(* CODESYS project Mk5 Aorta.library
   DefaultNamespace: _AORTA_
   Company: Atlas Copco
   Version: 2.0.0.0
   Title: Mk5 Aorta
   Author: Peter

Project tree, tasks and I/O mapping:
  libraries: Mk5 Definitions, 2.0.0.0 (Atlas Copco); Standard, * (System); SysMem, * (System); Mk5 Blackfin Libraries, 2.0.0.0 (Atlas Copco); Mk5 CANOpen Driver Interfaces, 2.0.0.0 (Atlas Copco); Mk5 CANOpen Driver Full, 2.0.0.0 (Atlas Copco); Mk5 IO and Protection System Interfaces, 2.0.0.0 (Atlas Copco); Mk5 Special IVL, 2.0.0.0 (Atlas Copco); Mk5 Lookup Tables Interfaces, 2.0.0.0 (Atlas Copco); Mk5 Display Texts Touch, 2.0.0.0 (Atlas Copco); Mk5 Drives Interfaces, 2.0.0.0 (Atlas Copco); Mk5 Tools Base Full, 2.0.0.0 (Atlas Copco); Mk5 CondensationPoint Interfaces, 2.0.0.0 (Atlas Copco); Mk5 Dryers Handler Interfaces, 2.0.0.0 (Atlas Copco); Mk5 Dryers Base Interfaces, 2.0.0.0 (Atlas Copco); Mk5 Retain Interfaces, 2.0.0.0 (Atlas Copco); Mk5 Special Functions interfaces, 2.0.0.0 (Atlas Copco); Mk5 StatusInfo Interfaces, 2.0.0.0 (Atlas Copco); Mk5 System Root, 2.0.0.0 (Atlas Copco); Mk5 Aorta Interfaces, 2.0.0.0 (Atlas Copco); Mk5 OD Interfaces, 2.0.0.0 (Atlas Copco); Mk5s Display Helpers Interfaces, 2.0.0.0 (Atlas Copco); Mk5s Display Base, 2.0.0.0 (Atlas Copco); Mk5s Display Definitions, 2.0.0.0 (Atlas Copco); Mk5 IO and Protection System Full, 2.0.0.0 (Atlas Copco); Mk5 CondensationPoint Full, 2.0.0.0 (Atlas Copco); Util, 3.5.18.0 (System); Mk5 SpeedControl Interfaces, 2.0.0.0 (Atlas Copco); Mk5 Display Constants, 2.0.0.0 (Atlas Copco); Mk5 ProtecSpec_Comon, 2.0.0.0 (Atlas Copco)
  Aorta/
    PrimaStuff/
      function block fbtCANOpenDriver_Aorta_Prima [ST]: mxInit, prpxValidData
      function block fbtAorta_Prima [ST]: mxInit, mxEnable, mxReset, mxResetCANOpenDriver, mxRun, mxPosition, mxHoming, mxDumpHomingSettings, prpxEnabled, mxWriteValue, prpdwPosition, mxConfigurationError
    Driver/
      CANOpenDriver/
        function block fbtCANOpenDriver_Aorta_Tri [ST]: mxInit, prpxValidData
        PDO Topic/
          Rx/
            function block fbtAorta_SW [ST]: prpx_2_OperationEnabled, prpx_0_ReadyToSwitchOn, prpx_5_QuickStop, prpx_9_Remote, prpx_4_VoltageEnabled, prpx_6_SwitchOnDisabled, prpx_12_SetpointInProcess, prpx_1_SwitchedOn, prpx_7_Warning, prpx_10_TargetReached, prpx_3_Fault, mbState
            function block fbtAorta_ActualPosition [ST]: prpdwPosition
            function block fbtAorta_ActualOperationMode [ST]: prpxHoming
            function block fbtAorta_ActualPosition_2Bytes [ST]: prpdwPosition
            function block fbtAorta_Alarm [ST]: prpwAlarm
            function block fbtAorta_SW_Trinamics [ST]: prpx_02_OperationEnabled, prpx_00_ReadyToSwitchOn, prpx_05_QuickStop, prpx_09_Remote, prpx_04_VoltageEnabled, prpx_06_SwitchOnDisabled, prpx_12_SetpointInProcess, prpx_01_SwitchedOn, prpx_07_Warning, prpx_10_TargetReached, prpx_03_Fault, mbState, prpx_14_MotorActive, prpx_15_Direction_Down, prpx_12_HomingMode_HomeAttained
            function block fbtAorta_ActualPosition_1 [ST]: prpdwPosition
          Tx/
            function block fbtAorta_CW [ST]: prpx_1_EnableVoltage, prpx_3_EnableOperation, prpx_0_SwitchOn, prpx_4_NewSetpoint, prpx_7_FaultReset, prpx_2_NoQuickStop, prpx_6_Relative, mxDisableOperation, mxShutDown
            function block fbtAorta_OperationMode [ST]: prpxHoming
            function block fbtAorta_HomingMode [ST]: prpbMode
            function block fbtAorta_TargetPosition [ST]: prpdwPosition
            function block fbtAorta_TargetPosition_2Bytes [ST]: prpdwPosition
            function block fbtAorta_Dummy_2Bytes [ST]: prpdwPosition
      function block fbtAorta_Trinamics [ST]: mxInit, mxPosition, dwMicroStepsMoved, mxHoming, mxReadStrokeLength, mxReadVendorID, prpxEnabled, mxEnable, mxReset, mxDisable, mxSettings, prpdwPosition, mxDumpSettings, mxCollectData, prpitfCANOpenDriver, mxForcedNMTReset, prpdiPCBTemp, prpdiHousingTemp, mxConfigurationError, prpwSW, prpdwError11Count, prpdwRequiredPosition, prpxDirection
      Settings/
        function block fbtAorta_AllSettings_Tri [ST]: mxInit, mxGetSDO
        function block fbtAorta_AllSettings_Pri [ST]: mxAdd, mxGetSDO, mxInit
      data type DS302_States
      data type Aorta_StateMachine
      data type Aorta_Errors
      data type Aorta_CycleStates
    AortaEngine/
      data type STR_Error
      function block fbtAortaSettingsDownloader [ST]: mxDownload, prpbActiveSubIndex, prpbStatus, prpxBusy, mxInit, prppDownloadError
      data type ENUM_AortaEngine_StateMain
      data type ENUM_AortaEngine_StateHoming
      data type ENUM_AortaEngine_StateOperating
      data type ENUM_AortaEngine_StateRetract
      function block fbtAortaEngine_Base [ST]: mxInit_SysPyLog, mxInit, mxInit_Output, mxLoadSettings, mxRun, mxHoming, mxOperating, mxEnable, mxRetract, mdiNextPosition, prppdiDebugPosition, prppdiDebugStroke_FullSteps, prppdiDebugStroke_MicroSteps, prppdiDebugStroke_Rotations, prppdiDebugError, prppdiDebugErrorPosition, prppdiDebugMicroStepsInMove, prppdiDebugRotDirection, prppdiDebugStallDetectPosition, prppdiDebugStallRetractDelta, prppdiDebugStallRetractPosition, prppdiStatusWord, prppdiDebugError11Counter, prpdwPosition, prpwError, mReset, mxOD3000Define, mxConfigurationError, prprLimitedPosition, prpxActive, prpxFixedPositionActive, prpxHomingActive, mxStartHoming, mxMoveToFixedPosition, prpdwHomingStrokeMS, prpxCANDriverError, mxCollectInfoSDO3000
      global variables GVL_AORTA
      data type ENUM_TimeUnit
      data type ENUM_AortaDownloader_States
      IVL/
        function block fbtIVL_STCPosition [ST]: mxIVL_Settings_Overwrite
    Special Alarm/
      function block fbtProtecSpec_STCValve [ST]: mxInitSpecial, mxLoadSettings, mwCheckProtection, prpitfProtectionInfo, prpxMoreInfo, mxReset, mxResolveMPLLinks
      function block fbtProtecSpec_STCValve_Info [ST]: mxGetMk5sData, mxSetMk5sData, mInit
  CoolPower/
    CANOpenDriver/
      function block fbtCANOpenDriver_CoolPower [ST]: mxInit, mxConfigPrep, mxSetAddress_NT, mxResetAddress
      function block fbtSDO_Series_CoolPower [ST]: mxGetSDO, mxInitList, prpbAddress
    PDO Topic/
      Rx/
        function block fbtCoolPower_ActualOperationMode [ST]: prpbOperationMode
        function block fbtCoolPower_ActualVelocity [ST]: prpdwVelocity
        function block fbtCoolPower_ActualPosition [ST]: prpdwPosition
        function block fbtCoolPower_SW [ST]: prpx_2_OperationEnabled, prpx_0_ReadyToSwitchOn, prpx_5_QuickStop, prpx_9_Remote, prpx_4_VoltageEnabled, prpx_6_SwitchOnDisabled, prpx_12_OMS1, prpx_1_SwitchedOn, prpx_7_Warning, prpx_10_TargetReached, prpx_3_Fault, mbState, prpx_8_Synchronized, prpx_11_InternalLimitActive, prpx_13_OMS2, prpx_15_ClosedLoop
        function block fbtCoolPower_DigitalInputs [ST]: mxGetInput
        function block fbtCoolPower_MaxMotorSpeed [ST]: prpdwMaxSpeed
        function block fbtCoolPower_RunningHours [ST]: prpdwRunningHours
        function block fbtCoolPower_SerialNumber_1_6 [ST]: prpdwSerial_1_6
        function block fbtCoolPower_SerialNumber_7_11 [ST]: prpdwSerial_7_11
      Tx/
        function block fbtCoolPower_CW [ST]: prpx_1_EnableVoltage, prpx_3_EnableOperation, prpx_0_SwitchOn, prpx_4_OMS1, prpx_7_FaultReset, prpx_2_NoQuickStop, prpx_8_Halt, prpx_5_OMS2, prpx_6_OMS3, prpx_9_OMS4
        function block fbtCoolPower_OperationMode [ST]: prpbOperationMode
        function block fbtCoolPower_TargetVelocity [ST]: prpdwVelocity
        function block fbtCoolPower_TargetPosition [ST]: prpdwPosition
        function block fbtCoolPower_DriveSubMode [ST]: prpx_0_ClosedLoop, prpx_1_VoS, prpx_2_Brake, prpx_3_CurrentReduction, prpx_5_Torque, prpx_6_BLDC
        function block fbtCoolPower_ProfileVelocity [ST]: prpdwVelocity
        function block fbtCoolPower_DigitalOutputs [ST]: mxSetOutput
      global variables GVL_NanoTecAddresses
    function block fbtCoolPower_NanoTec [ST]: prpbOperationMode, prpdwMaxSpeed, prpdwRunningHours, prpdwSpeed, prpulSerialNumber, prpxHalt, prpxIsOperational, prpbModel, prpdwTotalHours, mxDisable, mxEnable, mxInit, mxRun, mxReadOut, mxConfigure, mxReset, mxClean, mxResetCounter
  Oil Free Air/
    Offset/
      function block fbtOffsetsConditionalSetpointCalculation [ST]: mxInit, mxCollectInfoSDO3000, mxOD3000Define, mxRun, mxGetValueOffset
      function block fbtOffset [ST]: prprValue, mxGetInput, mxInit, prpbInputNumber, mxGetSubIndex, prpxZeroValue, mxGetPowerValue
    Conditional Setpoint/
      function block fbtConditionalSetpointCalculation [ST]: mxInit, mxInit_Output, mxRun, mxOD3000Define, mxCollectInfoSDO3000
      function block fbtInput_CondSetpoint_ERSetpoint [ST]: mxInit_ER, mxGetInput, prpxSwitchToER
      function block fbtIVL_CondSetpointTemp [ST]: mxSetOutput, prpwSDO, mxInit, prpbOffsetNumber, prpbOffsetNumberER, mxIVL_Settings_Overwrite
    Energy Recovery Regulation/
      function block fbtEnergyRecoveryRegulation [ST]: prprEnergyRecoverySetpointTemperature, mxInit, mxRun, prpxSwitchToER, mxOD3000Define, mxInit_Output
      data type ENUM_HeatQualityOffset
      function block fbtIVL_ERSetpointTemp [ST]: mxIVL_Settings_Overwrite
  Handler/
    function block fbtSTCHandler [ST]: mxGetSTCValve, mxInit, mxInit_Output, mxOD3000Define, mxRun, mxGetOptimalSERCalculation
  Industrial Air SER Calculation/
    function block fbtOptimalSERCalculation [ST]: mxInit, mxLoadSettings, mRun, prpiTemperature, prppdiDebugTemperature, mxInit_Output
    function block fbtIVL_OptimalSERTemp [ST]: mxIVL_Settings_Overwrite
*)

// Aorta/Driver/DS302_States
{attribute 'qualified_only'}
{attribute 'strict'}
TYPE DS302_States :
(
	bNoInfo,
	bNotReadyToSwitchOn,
	bSwitchOnDisabled,
	bReadyToSwitchOn,
	bSwitchedOn,
	bOperationEnabled,
	bQuickStopActive,
	bFault,
	bFaultReactionActive,
	bUnknown_Error,
	bWaitforReset
)BYTE;
END_TYPE

// Aorta/Driver/Aorta_StateMachine
{attribute 'qualified_only'}
{attribute 'strict'}
TYPE Aorta_StateMachine :
(
	bStart,
	bFlank,
	bFinish,
	bWait,
	bReadStroke,
	bMotorActive
)BYTE;
END_TYPE

// Aorta/Driver/Aorta_Errors
{attribute 'qualified_only'}
{attribute 'strict'}
TYPE Aorta_Errors :
(
	NoError							:= 0,
	Initiate_StartupTimeout			:= 1,
	Initiate_Fault					:= 2,
	Initiate_DumpSettings			:= 3,
	
	Homing_NotEnabled				:= 4,
	Homing_TimeOut					:= 5,
	Homing_FailedToGetStrokeLength	:= 6,
	Homing_RangeTooSmall			:= 7,
// 	Homing_Failed					:= 8,

	Position_NotEnabled				:= 9,
	Position_Stall					:= 10,
	Position_TimeOut				:= 11,
	Position_Retract				:= 12,
	Position_PI_Error				:= 13,
	STCValve_Active_No_Alarm		:= 14,
	CAN_Out							:= 100,
	StuckInErrorState				:= 101
)	BYTE
	:= NoError;
END_TYPE

// Aorta/Driver/Aorta_CycleStates
{attribute 'qualified_only'}
{attribute 'strict'}
TYPE Aorta_CycleStates :
(
	Idle,
	Send,
	TimeOut,
	StallDetected,
	StallHandling
	
);
END_TYPE

// Aorta/AortaEngine/STR_Error
TYPE STR_Error :
STRUCT
	tDelay			: TIME;
	tonDelay		: TON;
	bNotification	: BYTE;
END_STRUCT
END_TYPE

// Aorta/AortaEngine/ENUM_AortaEngine_StateMain
{attribute 'qualified_only'}
{attribute 'strict'}
TYPE ENUM_AortaEngine_StateMain :
(
	Enable,
	Homing,
	Operating,
	Retract,
	Reset,
	Error,
	CAN_Error,
	Valve_detached
);
END_TYPE

// Aorta/AortaEngine/ENUM_AortaEngine_StateHoming
{attribute 'qualified_only'}
{attribute 'strict'}
TYPE ENUM_AortaEngine_StateHoming :
(
	Start,
	Home,
	CheckRange,
	Retry
);
END_TYPE

// Aorta/AortaEngine/ENUM_AortaEngine_StateOperating
{attribute 'qualified_only'}
{attribute 'strict'}
TYPE ENUM_AortaEngine_StateOperating :
(
	GoToPosition,
	SetNextPosition,
	Wait
);
END_TYPE

// Aorta/AortaEngine/ENUM_AortaEngine_StateRetract
{attribute 'qualified_only'}
{attribute 'strict'}
TYPE ENUM_AortaEngine_StateRetract :
(
	SetRetractPosition,
	Retract
);
END_TYPE

// Aorta/AortaEngine/ENUM_TimeUnit
{attribute 'qualified_only'}
// {attribute 'strict'}
TYPE ENUM_TimeUnit :
(
	Millisecond	:= 0,
	Second		:= 1,
	Minute		:= 2,
	Hour		:= 3,
	Day			:= 4
)	BYTE;
END_TYPE

// Aorta/AortaEngine/ENUM_AortaDownloader_States
{attribute 'qualified_only'}
TYPE ENUM_AortaDownloader_States :
(
	findtype,
	select,
	download
);
END_TYPE

// Oil Free Air/Energy Recovery Regulation/ENUM_HeatQualityOffset
{attribute 'qualified_only'}
{attribute 'strict'}
TYPE ENUM_HeatQualityOffset :
(
	Not_used := 0,
	Input_IO,
	Minimal, 
	Medium, 
	Maximal	
	
)BYTE;
END_TYPE

// CoolPower/PDO Topic/GVL_NanoTecAddresses
{attribute 'qualified_only'}
VAR_GLOBAL CONSTANT
	SerialNumber1_6_Index 		: WORD := 16#2410;
	SerialNumber1_6_Subindex 	: BYTE := 1;
	SerialNumber7_11_Index 		: WORD := 16#2410;
	SerialNumber7_11_Subindex 	: BYTE := 2;
	RunningHours_Index			: WORD := 16#2410;
	RunningHours_Subindex		: BYTE := 3;
	TotalHours_Index			: WORD := 16#2410;
	TotalHours_Subindex			: BYTE := 4;
	MaxSpeed_Index				: WORD := 16#6080;
	MaxSpeed_Subindex			: BYTE := 0;
	Model_Index					: WORD := 16#2410;
	Model_Subindex				: BYTE := 5;
END_VAR

// Aorta/AortaEngine/GVL_AORTA
{attribute 'qualified_only'}
VAR_GLOBAL
	wControlRange 			: WORD := 10000;
	wControlRange01Percent 	: WORD := 1;  // same as above, but 0.1%
END_VAR

// Aorta/Driver/CANOpenDriver/PDO Topic/Tx/fbtAorta_CW
FUNCTION_BLOCK fbtAorta_CW EXTENDS fbtPDO_Word 
VAR_INPUT
END_VAR
VAR_OUTPUT
END_VAR
VAR
END_VAR

PROPERTY prpx_1_EnableVoltage : BOOL
SET
wData.1:=prpx_1_EnableVoltage;
END_SET
END_PROPERTY

PROPERTY prpx_3_EnableOperation : BOOL
SET
wData.3:=prpx_3_EnableOperation;
END_SET
END_PROPERTY

PROPERTY prpx_0_SwitchOn : BOOL
SET
wData.0:=prpx_0_SwitchOn;
END_SET
END_PROPERTY

PROPERTY prpx_4_NewSetpoint : BOOL
SET
wData.4:=prpx_4_NewSetpoint;
END_SET
END_PROPERTY

PROPERTY prpx_7_FaultReset : BOOL
SET
wData.7:=prpx_7_FaultReset;
END_SET
END_PROPERTY

PROPERTY prpx_2_NoQuickStop : BOOL
SET
wData.2:=prpx_2_NoQuickStop;
END_SET
END_PROPERTY

PROPERTY prpx_6_Relative : BOOL
SET
wData.6:=prpx_6_Relative;
END_SET
END_PROPERTY

METHOD mxDisableOperation : BOOL
VAR_INPUT
END_VAR
wData:=7;
END_METHOD

METHOD mxShutDown : BOOL
VAR_INPUT
END_VAR
wData:=6; //Shutdown aorta valve
END_METHOD

END_FUNCTION_BLOCK

// Aorta/Driver/CANOpenDriver/PDO Topic/Rx/fbtAorta_SW
FUNCTION_BLOCK fbtAorta_SW EXTENDS fbtPDO_Word 
VAR_INPUT
END_VAR
VAR_OUTPUT
END_VAR
VAR
END_VAR

PROPERTY prpx_2_OperationEnabled : BOOL
GET
prpx_2_OperationEnabled:=wData.2;
END_GET
END_PROPERTY

PROPERTY prpx_0_ReadyToSwitchOn : BOOL
GET
prpx_0_ReadyToSwitchOn:=wData.0;
END_GET
END_PROPERTY

PROPERTY prpx_5_QuickStop : BOOL
GET
prpx_5_QuickStop:=wData.5;
END_GET
END_PROPERTY

PROPERTY prpx_9_Remote : BOOL
GET
prpx_9_Remote:=wData.9;
END_GET
END_PROPERTY

PROPERTY prpx_4_VoltageEnabled : BOOL
GET
prpx_4_VoltageEnabled:=wData.4;
END_GET
END_PROPERTY

PROPERTY prpx_6_SwitchOnDisabled : BOOL
GET
prpx_6_SwitchOnDisabled:=wData.6;
END_GET
END_PROPERTY

PROPERTY prpx_12_SetpointInProcess : BOOL
GET
prpx_12_SetpointInProcess:=wData.12;
END_GET
END_PROPERTY

PROPERTY prpx_1_SwitchedOn : BOOL
GET
prpx_1_SwitchedOn:=wData.1;
END_GET
END_PROPERTY

PROPERTY prpx_7_Warning : BOOL
GET
prpx_7_Warning:=wData.7;
END_GET
END_PROPERTY

PROPERTY prpx_10_TargetReached : BOOL
GET
prpx_10_TargetReached:=wData.10;
END_GET
END_PROPERTY

PROPERTY prpx_3_Fault : BOOL
GET
prpx_3_Fault:=wData.3;
END_GET
END_PROPERTY

METHOD mbState : BYTE
VAR_INPUT
END_VAR
VAR
	wTmp : WORD;
END_VAR
wTmp := wData AND 16#000F;
CASE wTmp OF
0 : IF wData.6 THEN // wSW.prpx_6_SwitchOnDisabled 
		mbState := DS302_States.bSwitchOnDisabled;
	ELSE
		mbState := DS302_States.bNotReadyToSwitchOn;
	END_IF

1 : IF wData.5=1 AND wData.6=0 THEN
		mbState:= DS302_States.bReadyToSwitchOn;	
	ELSE
		mbState:=DS302_States.bUnknown_Error;
	END_IF

3 : IF wData.5=1 AND wData.6=0 THEN
		mbState:= DS302_States.bSwitchedOn;	
	ELSE
		mbState:=DS302_States.bUnknown_Error;
	END_IF

7 : IF wData.5=1 AND wData.6=0 THEN
		mbState:= DS302_States.bOperationEnabled;	
	ELSIF wData.5=0 AND wData.6=0 THEN
		mbState:= DS302_States.bQuickStopActive;	
	ELSE
		mbState:=DS302_States.bUnknown_Error;
	END_IF

8 : IF wData.6=0 THEN
		mbState:= DS302_States.bFault;	
	ELSE
		mbState:=DS302_States.bUnknown_Error;
	END_IF
		
16#F : IF wData.6=0 THEN
		mbState:= DS302_States.bFaultReactionActive;	
	ELSE
		mbState:=DS302_States.bUnknown_Error;
	END_IF
ELSE // case
			mbState:=DS302_States.bUnknown_Error;
END_CASE
END_METHOD

END_FUNCTION_BLOCK

// Aorta/Driver/CANOpenDriver/fbtCANOpenDriver_Aorta_Tri
FUNCTION_BLOCK fbtCANOpenDriver_Aorta_Tri EXTENDS fbtCANOpenDriver_Base
VAR_INPUT
END_VAR
VAR_OUTPUT
END_VAR
VAR
END_VAR

METHOD mxInit : BOOL
VAR_INPUT
	bCANAddress  			: BYTE;
END_VAR
eDriverState:=CAN_StateMachine.Idle;
bTheAddress := bCANAddress;

fbNMTCommands.mxInit(bAddress := bCANAddress);
END_METHOD

PROPERTY prpxValidData : BOOL
GET
prpxValidData:=TRUE;
END_GET
END_PROPERTY

END_FUNCTION_BLOCK

// Aorta/Driver/CANOpenDriver/PDO Topic/Tx/fbtAorta_OperationMode
FUNCTION_BLOCK fbtAorta_OperationMode EXTENDS fbtPDO_Byte
VAR_INPUT
END_VAR
VAR_OUTPUT
END_VAR
VAR
//	bMode : BYTE := 1;
END_VAR

PROPERTY prpxHoming : BOOL
SET
IF prpxHoming THEN
	bData := 6;
ELSE
	bData := 1; // pp
END_IF
END_SET
END_PROPERTY

END_FUNCTION_BLOCK

// Aorta/Driver/CANOpenDriver/PDO Topic/Tx/fbtAorta_HomingMode
FUNCTION_BLOCK fbtAorta_HomingMode EXTENDS fbtPDO_Byte
VAR_INPUT
END_VAR
VAR_OUTPUT
END_VAR
VAR
END_VAR

PROPERTY prpbMode : BYTE
SET
bData := prpbMode;
END_SET
END_PROPERTY

END_FUNCTION_BLOCK

// Aorta/Driver/CANOpenDriver/PDO Topic/Tx/fbtAorta_TargetPosition
FUNCTION_BLOCK fbtAorta_TargetPosition EXTENDS fbtPDO_DWORD
VAR_INPUT
END_VAR
VAR_OUTPUT
END_VAR
VAR
//	dwPosition : DWORD;
END_VAR

PROPERTY prpdwPosition : DWORD
SET
dwData := prpdwPosition;
END_SET
GET
prpdwPosition := dwData;
END_GET
END_PROPERTY

END_FUNCTION_BLOCK

// Aorta/Driver/CANOpenDriver/PDO Topic/Rx/fbtAorta_ActualPosition
FUNCTION_BLOCK fbtAorta_ActualPosition EXTENDS fbtPDO_DWORD
VAR_INPUT
END_VAR
VAR_OUTPUT
END_VAR
VAR
//	dwPosition : DWORD;
END_VAR

PROPERTY prpdwPosition : DWORD
GET
prpdwPosition:=dwData;
END_GET
END_PROPERTY

END_FUNCTION_BLOCK

// Aorta/Driver/CANOpenDriver/PDO Topic/Rx/fbtAorta_ActualOperationMode
FUNCTION_BLOCK fbtAorta_ActualOperationMode EXTENDS fbtPDO_Byte
VAR_INPUT
END_VAR
VAR_OUTPUT
END_VAR
VAR
//	bMode : BYTE := 1;
END_VAR

PROPERTY prpxHoming : BOOL
GET
IF bData = 6 THEN
	prpxHoming:=TRUE;
ELSE
	prpxHoming:=FALSE;
END_IF
END_GET
END_PROPERTY

END_FUNCTION_BLOCK

// Aorta/Driver/fbtAorta_Trinamics
FUNCTION_BLOCK fbtAorta_Trinamics
VAR
	bMyCANAddress			: BYTE;
	xStartLocal				: BOOL;
	
	fbCANOpen 				: fbtCANOpenDriver_Aorta_Tri;

	// dwBrand					: DWORD;
	
	Aorta_CW 				: fbtAorta_CW;
	Aorta_OperationMode 	: fbtAorta_OperationMode;
	Aorta_HomingMode 		: fbtAorta_HomingMode;
	Aorta_TargetPosition 	: fbtAorta_TargetPosition; 

	Aorta_SW				: fbtAorta_SW_Trinamics;
	Aorta_ActualPosition	: fbtAorta_ActualPosition;
	Aorta_ActualMode		: fbtAorta_ActualOperationMode;

	PCBTemp 				: fbtPDO_DWORD;
	HousingTemp             : fbtPDO_DWORD;

	wDownloadState			: WORD;
	xDownloadStart			: BOOL;
	wDownloadStateWait		: TON;
	
	Tp_CommandTimeOut		: TP;
	xStartTimeOut			: BOOL;
	bDriveState				: BYTE;
	
	bstate	 				: BYTE;
// position cycle
//	CycleTime 				: TON;
//	CycleState				: Aorta_CycleStates;
	TimeOut					: TON;

//	wCycleTime				: WORD;
	wPositioningTimeOut		: WORD;
	wHomingTimeOut			: WORD;

	xStartSend				: BOOL;
	xOK						: BOOL;
	wError					: WORD;
	// wNrStalls				: WORD;
	wDelayTime				: TON;
	SDO 					: fbtSDOCouple;
	
	dwPreviousPosition		: DWORD; // in 0.01%
	dwMicroStepsFactor	    : DWORD; // number of microsteps / 0.01%
	xDirection				: BOOL;

	dwError11Counter	: DWORD;
	
	xtmp1,xtmp2, xtmp3 : BOOL;
	xtmp10,xtmp20, xtmp30 : BOOL;
	
	//Debug
	xDebugTrigger			: BOOL := FALSE;
	
END_VAR

METHOD mxInit : BOOL
VAR_INPUT
	bCANAddress 			: BYTE;
//	wCycleTimeIn			: WORD;
	wPositioningTimeOutIn	: WORD;
	wHomingTimeOutIn		: WORD;

END_VAR
bMyCANAddress := bCANAddress;

wPositioningTimeOut		:= wPositioningTimeOutIn;
wHomingTimeOut			:= wHomingTimeOutIn;

Aorta_CW.mxActivateLog(sName := 'PDO Aorta CW',wLog:= eLogCodes._fixed_1);
Aorta_OperationMode.mxActivateLog(sName := 'PDO Aorta Operation Mode',wLog:= eLogCodes._fixed_1);
Aorta_HomingMode.mxActivateLog(sName := 'PDO Homing Mode',wLog:= eLogCodes._fixed_1);
Aorta_TargetPosition.mxActivateLog(sName := 'PDO Target Position',wLog:= eLogCodes._fixed_1);
Aorta_SW.mxActivateLog(sName := 'PDO Aorta SW',wLog:= eLogCodes._fixed_1);
Aorta_ActualPosition.mxActivateLog(sName := 'PDO Actual Position',wLog:= eLogCodes._fixed_1);
Aorta_ActualMode.mxActivateLog(sName := 'PDO Actual Mode',wLog:= eLogCodes._fixed_1);

SysPyLog.mxAdd(eCode := eLogCodes._fixed_1, pData := ADR(dwError11Counter),sNaam := 'Error11', eType := eLogTypes._dword);

fbCANOpen.mxInit(	bCANAddress 			:= bCANAddress);
	
fbCANOpen.mxClearPDOConfiguration();

fbCANOpen.mxAddTxPDOTopic(1, Aorta_CW);
fbCANOpen.mxAddTxPDOTopic(1, Aorta_OperationMode);
fbCANOpen.mxAddTxPDOTopic(1, Aorta_HomingMode);
fbCANOpen.mxAddTxPDOTopic(1, Aorta_TargetPosition);
fbCANOpen.mxBlockAutoRepeat(1, TRUE);
		
fbCANOpen.mxAddRxPDOTopic(1, Aorta_SW				, TRUE, 10000);
fbCANOpen.mxAddRxPDOTopic(1, Aorta_ActualPosition	, TRUE, 10000);
fbCANOpen.mxAddRxPDOTopic(1, Aorta_ActualMode		, TRUE, 10000);

fbCANOpen.mxAddRxPDOTopic(2, PCBTemp				, TRUE, 10000);
fbCANOpen.mxAddRxPDOTopic(2, HousingTemp			, TRUE, 10000);

TimeOut(IN:=FALSE);
END_METHOD

METHOD mxPosition : BOOL
VAR_INPUT
	dwPosition : DWORD; // in 0.01 %
	xRelative : BOOL;
END_VAR
VAR_IN_OUT
	xStart : BOOL;
END_VAR
VAR_OUTPUT
	xOk 			  : BOOL;
	wError 			  : WORD;
	dwMicroStepsInMove: DWORD; // number of microsteps moved by this action
END_VAR
IF xStart THEN
	xStart := FALSE;
	mxPosition := FALSE;
	bstate := Aorta_StateMachine.bStart;
	TimeOut(IN := FALSE);
	TimeOut(IN := TRUE,PT:= wPositioningTimeOut * T#1MS);
	wDelayTime(IN:=FALSE);
	
	xDirection :=  dwPosition > dwPreviousPosition; // false : down, true = up
	IF NOT prpxEnabled THEN
		xOK := FALSE;
		mxPosition := TRUE;
		wError := Aorta_Errors.Position_NotEnabled;
	END_IF
END_IF

CASE  bstate OF
	Aorta_StateMachine.bStart 	: 
		Aorta_HomingMode.prpbMode:=16#0;
		Aorta_OperationMode.prpxHoming:=FALSE;
		Aorta_CW.prpx_4_NewSetpoint:=0;
		Aorta_CW.prpx_6_Relative := xRelative;
		Aorta_TargetPosition.prpdwPosition := dwPosition;
		wDelayTime(IN:=TRUE,PT:=T#100MS);
		IF wDelayTime.Q THEN
			bstate := Aorta_StateMachine.bFlank;
		END_IF

	Aorta_StateMachine.bFlank 	: 
		Aorta_CW.prpx_4_NewSetpoint:=1;
		bstate := Aorta_StateMachine.bWait;
		wDelayTime(IN:=FALSE);	
		
	Aorta_StateMachine.bWait 	:
		xtmp1:= Aorta_SW.prpx_10_TargetReached;
		xtmp2:= Aorta_SW.prpx_14_MotorActive;
		xtmp3:= Aorta_SW.prpx_12_SetpointInProcess;
		wDelayTime(IN:=TRUE,PT:=T#100MS);
		IF wDelayTime.Q  THEN
			bState := Aorta_StateMachine.bMotorActive;
		END_IF

(*		
	Aorta_StateMachine.bWait :

		IF NOT Aorta_SW.prpx_12_SetpointInProcess THEN
			bState := Aorta_StateMachine.bFinish;
		END_IF
*)

	Aorta_StateMachine.bMotorActive	:
		IF NOT Aorta_SW.prpx_14_MotorActive THEN
			bState := Aorta_StateMachine.bFinish;
		END_IF


	Aorta_StateMachine.bFinish :
	
		xtmp10:= Aorta_SW.prpx_10_TargetReached;
		xtmp20:= Aorta_SW.prpx_14_MotorActive;
		xtmp30:= Aorta_SW.prpx_12_SetpointInProcess;
	
		IF Aorta_SW.prpx_10_TargetReached THEN
			dwMicroStepsInMove := dwMicroStepsMoved(xDirection := xDirection, dwPosition := dwPosition);
			dwPreviousPosition:=Aorta_ActualPosition.prpdwPosition;
			mxPosition := TRUE;
			xOK	:=	TRUE;
			wError := Aorta_Errors.NoError;
		ELSE
			mxPosition := TRUE;
			xOK := FALSE;
			wError := Aorta_Errors.Position_Stall;
			dwMicroStepsInMove := dwMicroStepsMoved(xDirection := xDirection, dwPosition := Aorta_ActualPosition.prpdwPosition);
			dwPreviousPosition:=Aorta_ActualPosition.prpdwPosition;
		END_IF

END_CASE

TimeOut(IN := TRUE,PT:= wPositioningTimeOut * T#1MS);
IF TimeOut.Q THEN
	dwError11Counter := dwError11Counter + 1;
	IF Aorta_SW.prpx_10_TargetReached THEN
		dwMicroStepsInMove := dwMicroStepsMoved(xDirection := xDirection, dwPosition := dwPosition);
		dwPreviousPosition := Aorta_ActualPosition.prpdwPosition;
		mxPosition := TRUE;
		xOK	:=	TRUE;
		wError := Aorta_Errors.NoError;
	ELSE
		mxPosition := TRUE;
		xOK := FALSE;
		wError := Aorta_Errors.Position_TimeOut;
		dwMicroStepsInMove := dwMicroStepsMoved(xDirection := xDirection, dwPosition := Aorta_ActualPosition.prpdwPosition);
		dwPreviousPosition:=Aorta_ActualPosition.prpdwPosition;
	END_IF
(*
	xOK := FALSE;
	mxPosition := TRUE;
	wError := Aorta_Errors.Position_TimeOut;
	xRotDirection:=xDirection;
	dwErrorPosition := Aorta_ActualPosition.prpdwPosition;
	dwMicroStepsInMove := dwMicroStepsMoved(xDirection := xDirection, dwPosition := dwErrorPosition);
	dwPreviousPosition:=dwErrorPosition;
*)

END_IF
END_METHOD

METHOD dwMicroStepsMoved : DWORD
VAR_INPUT
	xDirection : BOOL;
	dwPosition : DWORD;
END_VAR
IF xDirection THEN
	dwMicroStepsMoved := dwMicroStepsFactor * ( dwPosition - dwPreviousPosition);
ELSE
	dwMicroStepsMoved := dwMicroStepsFactor * ( dwPreviousPosition - dwPosition);
END_IF
END_METHOD

METHOD mxHoming : BOOL
VAR_IN_OUT
	xStart 		: BOOL;
END_VAR
VAR_OUTPUT
	dwStroke_microSteps	: DWORD;// number of microsteps
	dwStroke_FullSteps	: DWORD;// number of full steps
	rRotations			: REAL;	// real rotations
	xOk 				: BOOL;
	wError 				: WORD;
END_VAR
IF xStart THEN
	xStart := FALSE;
	mxHoming := FALSE;
	bstate := Aorta_StateMachine.bStart;
	
	wDelayTime(IN:=FALSE);

	TimeOut(IN := FALSE);
	TimeOut(IN := TRUE,PT:= wHomingTimeOut * T#1S);
	IF NOT prpxEnabled THEN
		xOK := FALSE;
		mxHoming := TRUE;
		wError := Aorta_Errors.Homing_NotEnabled;
	END_IF
END_IF

CASE  bstate OF
	Aorta_StateMachine.bStart 	: 
		Aorta_HomingMode.prpbMode:=16#FE;
		Aorta_OperationMode.prpxHoming:=TRUE;
		Aorta_CW.prpx_4_NewSetpoint:=0; // Stop homing
		Aorta_CW.prpx_6_Relative := FALSE;
		wDelayTime(IN:=TRUE,PT:=T#100MS);
		IF wDelayTime.Q THEN
			bstate := Aorta_StateMachine.bFlank;
		END_IF

	Aorta_StateMachine.bFlank 	: 
		Aorta_CW.prpx_4_NewSetpoint:=1; // Start homing
		bstate := Aorta_StateMachine.bWait;
		wDelayTime(IN:=FALSE);
		wDelayTime(IN:=TRUE,PT:=T#100MS);

	Aorta_StateMachine.bWait :
		wDelayTime(IN:=TRUE,PT:=T#100MS);
		IF wDelayTime.Q THEN
			bState := Aorta_StateMachine.bFinish;
		END_IF
		
	Aorta_StateMachine.bFinish 	: 
		IF Aorta_SW.prpx_12_HomingMode_HomeAttained THEN
			xStartLocal:=TRUE;
			bState := Aorta_StateMachine.bReadStroke;
		END_IF
		TimeOut(IN := TRUE,PT:= wHomingTimeOut * T#1S);
		IF TimeOut.Q THEN
			mxHoming := TRUE;
			xOK := FALSE;
			wError := Aorta_Errors.Homing_TimeOut;
		END_IF

	Aorta_StateMachine.bReadStroke :
		IF mxReadStrokeLength( xStart:=xStartLocal,xOK=>xOK,dwValue_MicroSteps =>dwStroke_microSteps,dwValue_FullSteps=>dwStroke_FullSteps, rValue=>rRotations) THEN
			IF NOT xOk THEN
				wError := Aorta_Errors.Homing_FailedToGetStrokeLength;
			END_IF
			dwPreviousPosition:=0;
			mxHoming:=TRUE;
		END_IF

END_CASE
END_METHOD

METHOD mxReadStrokeLength : BOOL
VAR_IN_OUT
	xStart 	: BOOL;
END_VAR
VAR_OUTPUT
	xOK 	: BOOL;
	dwValue_MicroSteps : DWORD; // microsteps
	dwValue_FullSteps : DWORD; // full 
	rValue	: REAL;  // rotations
END_VAR
VAR
	Value : ODItem;
END_VAR
IF xStart THEN
	SDO.mxMakeRead_Idx(bAddress := bMyCANAddress, wIndex := 16#20C2 , bSubIndex := 0);
END_IF
IF fbCANOpen.prpitfCANOpen_SDO.mxSDORead_Safe( itfSDOCouple := SDO, xStart := xStart, xOK => xOK) THEN
	Value:=SDO.prpDataReceived;
	dwValue_MicroSteps :=Value.dwValue;
	dwValue_FullSteps := SHR(Value.dwValue,8); // div by 256
	rValue:= DWORD_TO_REAL(dwValue_MicroSteps) / 51200;
	dwMicroStepsFactor:= dwValue_MicroSteps / GVL_Aorta.wControlRange; // per 0.1 %;
	mxReadStrokeLength:=TRUE;
END_IF
END_METHOD

METHOD mxReadVendorID : BOOL
VAR_IN_OUT
	xStart 	: BOOL;
END_VAR
VAR_OUTPUT
	dwVendorID : DWORD;
	xOK 		: BOOL;
END_VAR
VAR
	Value : ODItem;
END_VAR
IF xStart THEN
	SDO.mxMakeRead_Idx(bAddress := bMyCANAddress, wIndex := 16#1018 , bSubIndex := 1);
END_IF
IF fbCANOpen.prpitfCANOpen_SDO.mxSDORead_Safe( itfSDOCouple := SDO, xStart := xStart, xOK => xOK) THEN
	Value:=SDO.prpDataReceived;
	dwVendorID :=Value.dwValue;
	mxReadVendorID:=TRUE;
END_IF
END_METHOD

PROPERTY prpxEnabled : BOOL
GET
 prpxEnabled := Aorta_SW.mbState()= DS302_States.bOperationEnabled;
END_GET
END_PROPERTY

METHOD mxEnable : BOOL
VAR_IN_OUT
	xStart : BOOL;
END_VAR
VAR_OUTPUT
	xOK 	: BOOL; 
	wError 	: WORD;
END_VAR
mxEnable:=FALSE;
wError:=Aorta_Errors.NoError;

IF xStart THEN
	xStart:=FALSE;
	bDriveState:=Aorta_SW.mbState();
	// sometimes that CW seems not be different from the time before, but it was not seen by the device
	// with this action we make sure that the CW it send under all conditions.
//	Aorta_CW.prpxForceOneTimeSend := TRUE; => here it sometimes generates the sensing of 0 => error in aorta, for Aorta we make sure via the NMT machine that the DO was send
	Tp_CommandTimeOut(IN:=FALSE,PT:=T#4S); 
	xStartTimeOut:=TRUE;
END_IF

// Startup time-out timer, triggers if it takes too long to get this startup => problem
Tp_CommandTimeOut(IN:=xStartTimeOut,PT:=T#6S); // time to be defined
IF NOT Tp_CommandTimeOut.Q THEN
	wError:=Aorta_Errors.Initiate_StartupTimeout;
	mxEnable:=TRUE;
END_IF
xStartTimeOut:=FALSE;
// CANOpen drive states
CASE bDriveState OF
	DS302_States.bNoInfo 	 		 :
//		IF fbCANOpen.mxValidData THEN
			// ok we can start doing business :-)
		bDriveState:=Aorta_SW.mbState();
//		END_IF

	DS302_States.bNotReadyToSwitchOn 	: 
		bDriveState:=Aorta_SW.mbState();

	DS302_States.bSwitchOnDisabled  	: // transition 2 -> Ready Switch On
		// set appropriate bits to continue
		Aorta_CW.prpx_0_SwitchOn:=FALSE;
		Aorta_CW.prpx_1_EnableVoltage:=TRUE;
		Aorta_CW.prpx_2_NoQuickStop:=TRUE;
		Aorta_CW.prpx_3_EnableOperation:=FALSE;
//		fbSpeedTarget.mxForceZero();
		bDriveState:=Aorta_SW.mbState();
		
	DS302_States.bReadyToSwitchOn   	: // transition 3 -> Switched On
		// set appropriate bits to continue
		Aorta_CW.prpx_0_SwitchOn:=TRUE;
		Aorta_CW.prpx_1_EnableVoltage:=TRUE;
		Aorta_CW.prpx_2_NoQuickStop:=TRUE;
		Aorta_CW.prpx_3_EnableOperation:=FALSE;
//		fbSpeedTarget.mxForceZero();
		bDriveState:=Aorta_SW.mbState();

	DS302_States.bSwitchedOn 		  	: // transition 4 -> Operation Enabled
		// set appropriate bits to continue
		Aorta_CW.prpx_0_SwitchOn:=TRUE;
		Aorta_CW.prpx_1_EnableVoltage:=TRUE;
		Aorta_CW.prpx_2_NoQuickStop:=TRUE;
		Aorta_CW.prpx_3_EnableOperation:=TRUE;
//		fbSpeedTarget.mxForceZero();
		bDriveState:=Aorta_SW.mbState();
		
	DS302_States.bOperationEnabled  	: // stay at operation enabled
		Aorta_CW.prpx_0_SwitchOn:=TRUE;
		Aorta_CW.prpx_1_EnableVoltage:=TRUE;
		Aorta_CW.prpx_2_NoQuickStop:=TRUE;
		Aorta_CW.prpx_3_EnableOperation:=TRUE;
		xOK:=TRUE;
		mxEnable:=TRUE; 			// startup ok
		
	DS302_States.bQuickStopActive  	: // transition 16 -> Operation Enabled 
// start from QuickStop with speed:=0;
		Aorta_CW.prpx_0_SwitchOn:=TRUE;
		Aorta_CW.prpx_1_EnableVoltage:=TRUE;
		Aorta_CW.prpx_2_NoQuickStop:=TRUE;
		Aorta_CW.prpx_3_EnableOperation:=TRUE;
		bDriveState:=Aorta_SW.mbState();
		
	DS302_States.bFault, DS302_States.bFaultReactionActive, DS302_States.bUnknown_Error :
//		fbSpeedTarget.mxForceZero();
		Aorta_CW.mxClear();
		wError:= bDriveState;
		wError:= SHL(wError,8);
		wError:= wError + TO_BYTE(Aorta_Errors.Initiate_Fault);
		xOK:=FALSE;
		mxEnable:=TRUE;
		
		
		
END_CASE;
END_METHOD

METHOD mxReset : BOOL
VAR_INPUT
END_VAR
VAR_IN_OUT
	xStart : BOOL;
END_VAR
VAR_OUTPUT
	xOK 	: BOOL;
	wError 	: WORD;
END_VAR
mxReset:=FALSE;
wError:=0;

IF xStart THEN
	xStart:=FALSE;
	bDriveState:=Aorta_SW.mbState();
	Tp_CommandTimeOut(IN:=FALSE,PT:=T#4S); 
	xStartTimeOut:=TRUE;
END_IF

// Startup time-out timer, triggers if it takes too long to get this startup => problem
Tp_CommandTimeOut(IN:=xStartTimeOut,PT:=T#6S); // time to be defined
IF NOT Tp_CommandTimeOut.Q THEN
	wError:=1;
	mxReset:=TRUE;
END_IF
xStartTimeOut:=FALSE;
// CANOpen drive states
CASE bDriveState OF
	DS302_States.bFault, DS302_States.bFaultReactionActive, DS302_States.bUnknown_Error :
//		fbSpeedTarget.mxForceZero();
		Aorta_CW.mxClear();
		Aorta_CW.prpx_7_FaultReset:=TRUE;
	ELSE
		mxReset:=TRUE;
END_CASE;
END_METHOD

METHOD mxDisable : BOOL
VAR_IN_OUT
	xStart : BOOL;
END_VAR
VAR_OUTPUT
	xOK 	: BOOL; 
	wError 	: WORD;
END_VAR
mxDisable:=FALSE;
wError:=0;

IF xStart THEN
	xStart:=FALSE;
	bDriveState:=Aorta_SW.mbState();
	Tp_CommandTimeOut(IN:=FALSE,PT:=T#4S); 
	xStartTimeOut:=TRUE;
END_IF

// Startup time-out timer, triggers if it takes too long to get this stop => problem
Tp_CommandTimeOut(IN:=xStartTimeOut,PT:=T#4S); // time to be defined
IF NOT Tp_CommandTimeOut.Q THEN
	xOK:=FALSE;
	wError:=1;
	mxDisable:=TRUE;
	RETURN;
END_IF
xStartTimeOut:=FALSE;
CASE bDriveState OF
	DS302_States.bNoInfo 			 :
		bDriveState:=Aorta_SW.mbState();
	
	DS302_States.bNotReadyToSwitchOn 	: 
		bDriveState:=Aorta_SW.mbState();

 	DS302_States.bSwitchOnDisabled  	:	
			xOK:=FALSE;
			wError:=0;
			mxDisable:=TRUE;
			
	DS302_States.bReadyToSwitchOn 	: // transition 7 -> Switch On disabled
			Aorta_CW.mxClear(); 
			bDriveState:=Aorta_SW.mbState();
	
	DS302_States.bSwitchedOn 		  	: // transition 10 -> Switch On disabled
			Aorta_CW.mxClear();
			bDriveState:=Aorta_SW.mbState();
		
	DS302_States.bOperationEnabled  	: // transition 5 -> Switched on
			Aorta_CW.mxDisableOperation();
			bDriveState:=Aorta_SW.mbState();
			
	DS302_States.bQuickStopActive  	: // transition 12 
			Aorta_CW.mxClear();
			bDriveState:=Aorta_SW.mbState();

	DS302_States.bFault, DS302_States.bFaultReactionActive, DS302_States.bUnknown_Error :
			Aorta_CW.mxClear();
			mxDisable:=TRUE;
	END_CASE;
END_METHOD

METHOD mxSettings : BOOL
VAR
	TmpItem	: ODItem;
END_VAR
END_METHOD

PROPERTY prpdwPosition : DWORD
GET
prpdwPosition := Aorta_ActualPosition.prpdwPosition;
END_GET
END_PROPERTY

METHOD mxDumpSettings : BOOL
VAR_INPUT
	itfSettings : itf_SDO_FullList;
END_VAR
VAR_OUTPUT
	xOK : BOOL;
END_VAR
VAR_IN_OUT
	xStart : BOOL;
END_VAR
IF xStart THEN
	xStart := FALSE;
	wDownloadState := 1;
	wDownloadStateWait(IN:=FALSE,PT:=T#500MS);
END_IF

CASE wDownloadState OF

	1:	fbCANOpen.prpitfNMTCommands.mxResetNode();
		wDownloadStateWait(IN:=TRUE,PT:=T#500MS);
		wDownloadState := 2;
	
	2 : wDownloadStateWait(IN:=TRUE,PT:=T#500MS);
		IF wDownloadStateWait.Q THEN
			wDownloadState := 3;
			xDownloadStart := TRUE;
		END_IF

	3 :  mxDumpSettings:=fbCANOpen.prpitfCANOpen_SDO.mxWriteFullList(	xstart:= xDownloadStart, bMyCANAddress := bMyCANAddress, itfList := itfSettings, xOK=>xOK);

END_CASE
END_METHOD

METHOD mxCollectData : BOOL
VAR_INPUT
	itfData : itf_SDO_FullList;
END_VAR
VAR_OUTPUT
	xOK : BOOL;
END_VAR
VAR_IN_OUT
	xStart : BOOL;
END_VAR
mxCollectData:=fbCANOpen.prpitfCANOpen_SDO.mxReadFullList(	xstart:= xStart, 	
															bMyCANAddress := bMyCANAddress,
															itfList := itfData,
															xOK=>xOK);
END_METHOD

PROPERTY prpitfCANOpenDriver : itf_canopendriver
GET
prpitfCANOpenDriver:=fbCANOpen;
END_GET
END_PROPERTY

METHOD mxForcedNMTReset : BOOL
VAR_INPUT
END_VAR
fbCANOpen.prpitfNMTCommands.mxResetNode();
END_METHOD

PROPERTY prpdiPCBTemp : DINT
GET
VAR
	ditemp : DINT;
END_VAR
sysmemcpy(ADR(ditemp),PCBTemp.prppbRaw,PCBTemp.prpbsize);
prpdiPCBTemp:=ditemp;
END_GET
END_PROPERTY

PROPERTY prpdiHousingTemp : DINT
GET
VAR
	ditemp : DINT;
END_VAR
sysmemcpy(ADR(ditemp),HousingTemp.prppbRaw,HousingTemp.prpbsize);
prpdiHousingTemp:=ditemp;
END_GET
END_PROPERTY

METHOD mxConfigurationError : BOOL
VAR_OUTPUT
	bError : BYTE;
END_VAR
mxConfigurationError := FALSE;
IF fbCANOpen.prpbConfigError <> 0 THEN
	mxConfigurationError := TRUE;
	bError := fbCANOpen.prpbConfigError;
END_IF
END_METHOD

PROPERTY prpwSW : WORD
GET
prpwSW:=Aorta_SW.prpwRawData;
END_GET
END_PROPERTY

PROPERTY prpdwError11Count : DWORD
GET
prpdwError11Count:=dwError11Counter;
END_GET
END_PROPERTY

PROPERTY prpdwRequiredPosition : DWORD
GET
prpdwRequiredPosition:=Aorta_TargetPosition.prpdwPosition;
END_GET
END_PROPERTY

PROPERTY prpxDirection : BOOL
GET
//down => false
//up => true
prpxDirection := xDirection;
END_GET
END_PROPERTY

END_FUNCTION_BLOCK

// Aorta/Driver/CANOpenDriver/PDO Topic/Rx/fbtAorta_SW_Trinamics
FUNCTION_BLOCK fbtAorta_SW_Trinamics EXTENDS fbtPDO_Word 
VAR_INPUT
END_VAR
VAR_OUTPUT
END_VAR
VAR
END_VAR

PROPERTY prpx_02_OperationEnabled : BOOL
GET
prpx_02_OperationEnabled:=wData.2;
END_GET
END_PROPERTY

PROPERTY prpx_00_ReadyToSwitchOn : BOOL
GET
prpx_00_ReadyToSwitchOn:=wData.0;
END_GET
END_PROPERTY

PROPERTY prpx_05_QuickStop : BOOL
GET
prpx_05_QuickStop:=wData.5;
END_GET
END_PROPERTY

PROPERTY prpx_09_Remote : BOOL
GET
prpx_09_Remote:=wData.9;
END_GET
END_PROPERTY

PROPERTY prpx_04_VoltageEnabled : BOOL
GET
prpx_04_VoltageEnabled:=wData.4;
END_GET
END_PROPERTY

PROPERTY prpx_06_SwitchOnDisabled : BOOL
GET
prpx_06_SwitchOnDisabled:=wData.6;
END_GET
END_PROPERTY

PROPERTY prpx_12_SetpointInProcess : BOOL
GET
prpx_12_SetpointInProcess:=wData.12;
END_GET
END_PROPERTY

PROPERTY prpx_01_SwitchedOn : BOOL
GET
prpx_01_SwitchedOn:=wData.1;
END_GET
END_PROPERTY

PROPERTY prpx_07_Warning : BOOL
GET
prpx_07_Warning:=wData.7;
END_GET
END_PROPERTY

PROPERTY prpx_10_TargetReached : BOOL
GET
prpx_10_TargetReached:=wData.10;
END_GET
END_PROPERTY

PROPERTY prpx_03_Fault : BOOL
GET
prpx_03_Fault:=wData.3;
END_GET
END_PROPERTY

METHOD mbState : BYTE
VAR_INPUT
END_VAR
VAR
	wTmp : WORD;
END_VAR
wTmp := wData AND 16#000F;
CASE wTmp OF
0 : IF wData.6 THEN // wSW.prpx_6_SwitchOnDisabled 
		mbState := DS302_States.bSwitchOnDisabled;
	ELSE
		mbState := DS302_States.bNotReadyToSwitchOn;
	END_IF

1 : IF wData.5=1 AND wData.6=0 THEN
		mbState:= DS302_States.bReadyToSwitchOn;	
	ELSE
		mbState:=DS302_States.bUnknown_Error;
	END_IF

3 : IF wData.5=1 AND wData.6=0 THEN
		mbState:= DS302_States.bSwitchedOn;	
	ELSE
		mbState:=DS302_States.bUnknown_Error;
	END_IF

7 : IF wData.5=1 AND wData.6=0 THEN
		mbState:= DS302_States.bOperationEnabled;	
	ELSIF wData.5=0 AND wData.6=0 THEN
		mbState:= DS302_States.bQuickStopActive;	
	ELSE
		mbState:=DS302_States.bUnknown_Error;
	END_IF

8 : IF wData.6=0 THEN
		mbState:= DS302_States.bFault;	
	ELSE
		mbState:=DS302_States.bUnknown_Error;
	END_IF
		
16#F : IF wData.6=0 THEN
		mbState:= DS302_States.bFaultReactionActive;	
	ELSE
		mbState:=DS302_States.bUnknown_Error;
	END_IF
ELSE // case
		mbState:=DS302_States.bUnknown_Error;
END_CASE
END_METHOD

PROPERTY prpx_14_MotorActive : BOOL
GET
prpx_14_MotorActive:=wData.14;
END_GET
END_PROPERTY

PROPERTY prpx_15_Direction_Down : BOOL
GET
prpx_15_Direction_Down:=wData.15;
END_GET
END_PROPERTY

PROPERTY prpx_12_HomingMode_HomeAttained : BOOL
GET
prpx_12_HomingMode_HomeAttained:=wData.12;
END_GET
END_PROPERTY

END_FUNCTION_BLOCK

// Aorta/PrimaStuff/fbtCANOpenDriver_Aorta_Prima
FUNCTION_BLOCK fbtCANOpenDriver_Aorta_Prima EXTENDS fbtCANOpenDriver_Base
VAR_INPUT
END_VAR
VAR_OUTPUT
END_VAR
VAR
END_VAR

METHOD mxInit : BOOL
VAR_INPUT
	bCANAddress  			: BYTE;
END_VAR
eDriverState:=CAN_StateMachine.Idle;
bTheAddress := bCANAddress;

fbNMTCommands.mxInit(bAddress := bCANAddress);
END_METHOD

PROPERTY prpxValidData : BOOL
GET
prpxValidData:=TRUE;
END_GET
END_PROPERTY

END_FUNCTION_BLOCK

// Aorta/PrimaStuff/fbtAorta_Prima
FUNCTION_BLOCK fbtAorta_Prima
VAR_INPUT
END_VAR
VAR_OUTPUT
END_VAR
VAR
	bMyCANAddress			: BYTE;
	xStartLocal				: BOOL;
	
	fbCANOpen 				: fbtCANOpenDriver_Aorta_Prima;
//	fbSDOs					: fbtSDOCouple;
	
	Aorta_CW 				: fbtAorta_CW;
	Aorta_OperationMode 	: fbtAorta_OperationMode;
	Aorta_HomingMode 		: fbtAorta_HomingMode;
	Aorta_TargetPosition 	: fbtAorta_TargetPosition_2Bytes; 

	Aorta_SW				: fbtAorta_SW;
	Aorta_ActualPosition	: fbtAorta_ActualPosition_2Bytes;
	Aorta_ActualMode		: fbtAorta_ActualOperationMode;
	Aorta_Alarm				: fbtAorta_Alarm;
	Aorta_dummy				: fbtAorta_Dummy_2Bytes;
	

	Tp_CommandTimeOut		: TP;
	xStartTimeOut			: BOOL;
	bDriveState				: BYTE;
	wDelayTime				: TON;
	
	bstate	 				: BYTE;
//	Setting2Download		: SingleSetting;

	SDO 					: fbtSDOCouple;
	OneSDO					: SingleFullSDO;
	
END_VAR

METHOD mxInit : BOOL
VAR_INPUT
	bCANAddress : BYTE;
END_VAR
bMyCANAddress := bCANAddress;

fbCANOpen.mxInit(bCANAddress 			:= bCANAddress);

fbCANOpen.mxClearPDOConfiguration();

fbCANOpen.mxAddTxPDOTopic(1,Aorta_CW);
fbCANOpen.mxAddTxPDOTopic(1,Aorta_OperationMode);
fbCANOpen.mxAddTxPDOTopic(1,Aorta_HomingMode);
fbCANOpen.mxAddTxPDOTopic(1,Aorta_TargetPosition);
fbCANOpen.mxAddTxPDOTopic(1,Aorta_dummy);

fbCANOpen.mxAddRxPDOTopic(1,Aorta_SW			, TRUE, 10000);
fbCANOpen.mxAddRxPDOTopic(1,Aorta_ActualPosition, TRUE, 10000);
fbCANOpen.mxAddRxPDOTopic(1,Aorta_ActualMode	, TRUE, 10000);
fbCANOpen.mxAddRxPDOTopic(1,Aorta_Alarm			, TRUE, 10000);
END_METHOD

METHOD mxEnable : BOOL
VAR_INPUT
END_VAR
VAR_IN_OUT
	xStart : BOOL;
END_VAR
VAR_OUTPUT
	xOK 	: BOOL;
	wError 	: WORD;
END_VAR
mxEnable:=FALSE;
wError:=0;

IF xStart THEN
	xStart:=FALSE;
//	IF fbCANOpen.mxValidData 	THEN bDriveState:=Aorta_SW.mbState();
//							ELSE bDriveState:=bAorta_NoInfo; END_IF
	bDriveState:=Aorta_SW.mbState();
	Tp_CommandTimeOut(IN:=FALSE,PT:=T#4S); 
	Aorta_CW.mxClear();
	xStartTimeOut:=TRUE;
END_IF

// Startup time-out timer, triggers if it takes too long to get this startup => problem
Tp_CommandTimeOut(IN:=xStartTimeOut,PT:=T#6S); // time to be defined
IF NOT Tp_CommandTimeOut.Q THEN
	wError:=1;
	mxEnable:=TRUE;
END_IF
xStartTimeOut:=FALSE;
// CANOpen drive states
CASE bDriveState OF
	DS302_States.bNoInfo 	 		 :
//		IF fbCANOpen.mxValidData THEN
			// ok we can start doing business :-)
		bDriveState:=Aorta_SW.mbState();
//		END_IF

	DS302_States.bNotReadyToSwitchOn 	: 
		bDriveState:=Aorta_SW.mbState();

	DS302_States.bSwitchOnDisabled  	: // transition 2 -> Ready Switch On
		// set appropriate bits to continue
		Aorta_CW.prpx_0_SwitchOn:=FALSE;
		Aorta_CW.prpx_1_EnableVoltage:=TRUE;
		Aorta_CW.prpx_2_NoQuickStop:=TRUE;
		Aorta_CW.prpx_3_EnableOperation:=FALSE;
//		fbSpeedTarget.mxForceZero();
		bDriveState:=Aorta_SW.mbState();
		
	DS302_States.bReadyToSwitchOn   	: // transition 3 -> Switched On
		// set appropriate bits to continue
		Aorta_CW.prpx_0_SwitchOn:=TRUE;
		Aorta_CW.prpx_1_EnableVoltage:=TRUE;
		Aorta_CW.prpx_2_NoQuickStop:=TRUE;
		Aorta_CW.prpx_3_EnableOperation:=FALSE;
//		fbSpeedTarget.mxForceZero();
		bDriveState:=Aorta_SW.mbState();

	DS302_States.bSwitchedOn 		  	: // transition 4 -> Operation Enabled
		// set appropriate bits to continue
		Aorta_CW.prpx_0_SwitchOn:=TRUE;
		Aorta_CW.prpx_1_EnableVoltage:=TRUE;
		Aorta_CW.prpx_2_NoQuickStop:=TRUE;
		Aorta_CW.prpx_3_EnableOperation:=TRUE;
//		fbSpeedTarget.mxForceZero();
		bDriveState:=Aorta_SW.mbState();
		
	DS302_States.bOperationEnabled  	: // stay at operation enabled
		Aorta_CW.prpx_0_SwitchOn:=TRUE;
		Aorta_CW.prpx_1_EnableVoltage:=TRUE;
		Aorta_CW.prpx_2_NoQuickStop:=TRUE;
		Aorta_CW.prpx_3_EnableOperation:=TRUE;
//		fbSpeedTarget.mxReleaseSpeed();
		mxEnable:=TRUE; 			// startup ok
		
	DS302_States.bQuickStopActive  	: // transition 16 -> Operation Enabled 
// start from QuickStop with speed:=0;
		Aorta_CW.prpx_0_SwitchOn:=TRUE;
		Aorta_CW.prpx_1_EnableVoltage:=TRUE;
		Aorta_CW.prpx_2_NoQuickStop:=TRUE;
		Aorta_CW.prpx_3_EnableOperation:=TRUE;
		bDriveState:=Aorta_SW.mbState();
//		fbSpeedTarget.mxForceZero();

//	bDriveState_FaultReactionActive :
//		bDriveState:=fbSW.mbState();
		
	DS302_States.bFault, DS302_States.bFaultReactionActive, DS302_States.bUnknown_Error :
//		fbSpeedTarget.mxForceZero();
		Aorta_CW.mxClear();
		wError:=2;
		mxEnable:=TRUE;
END_CASE;
END_METHOD

METHOD mxReset : BOOL
VAR_INPUT
END_VAR
VAR_IN_OUT
	xStart : BOOL;
END_VAR
VAR_OUTPUT
	xOK 	: BOOL;
	wError 	: WORD;
END_VAR
mxReset:=FALSE;
wError:=0;

IF xStart THEN
	xStart:=FALSE;
	bDriveState:=Aorta_SW.mbState();
	Tp_CommandTimeOut(IN:=FALSE,PT:=T#4S); 
	xStartTimeOut:=TRUE;
END_IF

// Startup time-out timer, triggers if it takes too long to get this startup => problem
Tp_CommandTimeOut(IN:=xStartTimeOut,PT:=T#6S); // time to be defined
IF NOT Tp_CommandTimeOut.Q THEN
	wError:=1;
	mxReset:=TRUE;
END_IF
xStartTimeOut:=FALSE;
// CANOpen drive states
CASE bDriveState OF
	DS302_States.bFault, DS302_States.bFaultReactionActive, DS302_States.bUnknown_Error :
//		fbSpeedTarget.mxForceZero();
		Aorta_CW.mxClear();
		Aorta_CW.prpx_7_FaultReset:=TRUE;
	ELSE
		mxReset:=TRUE;
END_CASE;
END_METHOD

METHOD mxResetCANOpenDriver : BOOL
VAR_INPUT
END_VAR
fbCANOpen.mxReset();
END_METHOD

METHOD mxRun : BOOL
VAR_INPUT
END_VAR
fbCanOpen.mxRun();
END_METHOD

METHOD mxPosition : BOOL
VAR_INPUT
	dwPosition : DWORD; // in 0.01 %
END_VAR
VAR_IN_OUT
	xStart : BOOL;
END_VAR
VAR_OUTPUT
	xOk 	: BOOL;
	wError 	: WORD;
END_VAR
IF xStart THEN
	xStart := FALSE;
	mxPosition := FALSE;
	bstate := Aorta_StateMachine.bStart;
	IF NOT prpxEnabled THEN
		xOK := FALSE;
		mxPosition := TRUE;
		wError := Aorta_Errors.Position_NotEnabled;
	END_IF
END_IF

CASE  bstate OF
	
	Aorta_StateMachine.bStart 	: 
		Aorta_HomingMode.prpbMode:=16#0;
		Aorta_OperationMode.prpxHoming:=FALSE;
		Aorta_CW.prpx_4_NewSetpoint:=0;
		Aorta_TargetPosition.prpdwPosition := dwPosition;
		bstate := Aorta_StateMachine.bWait;
		wDelayTime(IN:=FALSE);
		wDelayTime(IN:=TRUE,PT:=T#120MS);

	Aorta_StateMachine.bWait :
		wDelayTime(IN:=TRUE,PT:=T#120MS);
		IF wDelayTime.Q THEN
			bState := Aorta_StateMachine.bFinish;
		END_IF
		
	Aorta_StateMachine.bFinish 	: 
		Aorta_CW.prpx_4_NewSetpoint:=1;
		IF Aorta_SW.prpx_12_SetpointInProcess THEN
			mxPosition := TRUE;
			xOK	:=	TRUE;
			wError := 0;
		END_IF

END_CASE
END_METHOD

METHOD mxHoming : BOOL
VAR_IN_OUT
	xStart : BOOL;
END_VAR
VAR_OUTPUT
	xOk 	: BOOL;
	wError 	: WORD;
END_VAR
IF xStart THEN
	xStart := FALSE;
	mxHoming := FALSE;
	bstate := Aorta_StateMachine.bStart;
	IF NOT prpxEnabled THEN
		xOK := FALSE;
		mxHoming := TRUE;
		wError := Aorta_Errors.Homing_NotEnabled;
	END_IF
END_IF

CASE  bstate OF
	
	Aorta_StateMachine.bStart 	: 
		Aorta_HomingMode.prpbMode:=1;
		Aorta_OperationMode.prpxHoming:=TRUE;
		Aorta_CW.prpx_4_NewSetpoint:=0;
		bstate := Aorta_StateMachine.bWait;
		wDelayTime(IN:=FALSE);
		wDelayTime(IN:=TRUE,PT:=T#120MS);

	Aorta_StateMachine.bWait :
		wDelayTime(IN:=TRUE,PT:=T#120MS);
		IF wDelayTime.Q THEN
			bState := Aorta_StateMachine.bFinish;
		END_IF
	
	Aorta_StateMachine.bFinish 	: 
		Aorta_CW.prpx_4_NewSetpoint:=1;
		IF Aorta_SW.prpx_12_SetpointInProcess THEN
			mxHoming := TRUE;
			xOK	:=	TRUE;
			wError := 0;
		END_IF

END_CASE
END_METHOD

METHOD mxDumpHomingSettings : BOOL
VAR_INPUT
	itfSettings : itf_SDO_FullList;
END_VAR
VAR_OUTPUT
	xOK : BOOL;
END_VAR
VAR_IN_OUT
	xStart : BOOL;
END_VAR
mxDumpHomingSettings:=TRUE;
END_METHOD

PROPERTY prpxEnabled : BOOL
GET
 prpxEnabled := Aorta_SW.mbState()= DS302_States.bOperationEnabled;
END_GET
END_PROPERTY

METHOD mxWriteValue : BOOL
VAR_INPUT
	Data : SingleFullSDO;
END_VAR
VAR_IN_OUT
	xStart : BOOL;
END_VAR
VAR_OUTPUT
	xOK : BOOL;
END_VAR
IF xStart THEN
	OneSDO := Data;
	SDO.mxMakeWriteFull(bAddress := bMyCANAddress, pSDO := ADR(Data));
END_IF
mxWriteValue := fbCANOpen.prpitfCANOpen_SDO.mxSDOWrite_Safe(itfSDOCouple := SDO, xStart := xStart, xOK => xOK);
END_METHOD

PROPERTY prpdwPosition : DWORD
GET
prpdwPosition := Aorta_ActualPosition.prpdwPosition;
END_GET
END_PROPERTY

METHOD mxConfigurationError : BOOL
VAR_OUTPUT
	bError : BYTE;
END_VAR
mxConfigurationError := FALSE;
IF fbCANOpen.prpbConfigError <> 0 THEN
	mxConfigurationError := TRUE;
	bError := fbCANOpen.prpbConfigError;
END_IF
END_METHOD

END_FUNCTION_BLOCK

// Aorta/Driver/CANOpenDriver/PDO Topic/Tx/fbtAorta_TargetPosition_2Bytes
FUNCTION_BLOCK fbtAorta_TargetPosition_2Bytes EXTENDS fbtPDO_WORD
VAR_INPUT
END_VAR
VAR_OUTPUT
END_VAR
VAR
//	wPosition : DWORD;
END_VAR

PROPERTY prpdwPosition : DWORD
SET
wData := DWORD_TO_WORD(prpdwPosition);
END_SET
END_PROPERTY

END_FUNCTION_BLOCK

// Aorta/Driver/CANOpenDriver/PDO Topic/Rx/fbtAorta_ActualPosition_2Bytes
FUNCTION_BLOCK fbtAorta_ActualPosition_2Bytes EXTENDS fbtPDO_WORD
VAR_INPUT
END_VAR
VAR_OUTPUT
END_VAR
VAR
//	dwPosition : DWORD;
END_VAR

PROPERTY prpdwPosition : DWORD
GET
prpdwPosition:=wData;
END_GET
END_PROPERTY

END_FUNCTION_BLOCK

// Aorta/Driver/CANOpenDriver/PDO Topic/Rx/fbtAorta_Alarm
FUNCTION_BLOCK fbtAorta_Alarm EXTENDS fbtPDO_WORD
VAR_INPUT
END_VAR
VAR_OUTPUT
END_VAR
VAR
//	dwPosition : DWORD;
END_VAR

PROPERTY prpwAlarm : DWORD
GET
prpwAlarm:=wData;
END_GET
END_PROPERTY

END_FUNCTION_BLOCK

// Aorta/Driver/CANOpenDriver/PDO Topic/Tx/fbtAorta_Dummy_2Bytes
FUNCTION_BLOCK fbtAorta_Dummy_2Bytes EXTENDS fbtPDO_WORD
VAR_INPUT
END_VAR
VAR_OUTPUT
END_VAR
VAR
//	wPosition : DWORD;
END_VAR

PROPERTY prpdwPosition : DWORD
SET
wData := DWORD_TO_WORD(prpdwPosition);
END_SET
END_PROPERTY

END_FUNCTION_BLOCK

// CoolPower/CANOpenDriver/fbtCANOpenDriver_CoolPower
FUNCTION_BLOCK fbtCANOpenDriver_CoolPower EXTENDS fbtCANOpenDriver_Base
VAR_INPUT
END_VAR
VAR_OUTPUT
END_VAR
VAR
	bLSS_State				: BYTE;
	bCurrentAddress 		: BYTE;
	bConnectionAttempts		: BYTE;
	Vendor		: fbtSDOCouple;
	Product		: fbtSDOCouple;
	Revision	: fbtSDOCouple;
	Serial		: fbtSDOCouple;
	tonReadDelay	: TON;
END_VAR
VAR CONSTANT
	bSendSetAddress 		: BYTE := 0;
	bCheckSetAddress		: BYTE := 1;
	bSendDefaultAddress 	: BYTE := 2;
	bCheckDefaultAddress	: BYTE := 3;
	bWriteAddress			: BYTE := 4;
	bSaveAddress			: BYTE := 5;
	bReset					: BYTE := 6;
	bLSSConfig				: BYTE := 7;
	bLSSRequestAddress		: BYTE := 8;
	bLSSReadAddress			: BYTE := 9;
	bLSSWait				: BYTE := 10;
	bResetAddress			: BYTE := 11;
	bAddressSet				: BYTE := 99;
END_VAR

METHOD mxInit : BOOL
VAR_INPUT
	bCANAddress  			: BYTE;
END_VAR
eDriverState		:= CAN_StateMachine.Idle;
bTheAddress 		:= bCANAddress;
bConnectionAttempts := 0;
END_METHOD

METHOD mxConfigPrep : BOOL
VAR_INPUT
END_VAR
mxConfigPrep := FALSE;
CASE eDriverState OF
	CAN_StateMachine.Reset :
	// this is needed to get the PDO's running
		fbNMTCommands.mxResetNode();
		eDriverState:=CAN_StateMachine.Idle;

	CAN_StateMachine.Idle :
		xStart:=TRUE;
		fbNMTCommands.mxNodeGuardCheck_Reset();
		eDriverState:=CAN_StateMachine.Init;
		
	CAN_StateMachine.Init 	: 
		IF fbNMTCommands.mxChangeState(eState := NMT_States.PreOperational, xStart:=xStart) THEN
			IF fbNMTCommands.prpeNodeState = NMT_States.PreOperational THEN
				eDriverState:=CAN_StateMachine.Configure;
				ELSE
				eDriverState:=CAN_StateMachine.Error;
			END_IF
		END_IF

	CAN_StateMachine.Configure:
		IF  fbNMTCommands.prpeNodeState = NMT_States.PreOperational THEN
			mxConfigPrep := TRUE;
		ELSE
			eDriverState:=CAN_StateMachine.Error;
		END_IF;
		
	CAN_StateMachine.Stopped :
		fbNMTCommands.mxResetNode();

	CAN_StateMachine.Error 			:
		eDriverState:=CAN_StateMachine.Idle; // reset the driver automatically
//		fbRxPDO1.mxClear();
ELSE
	eDriverState := CAN_StateMachine.Idle;
END_CASE
END_METHOD

METHOD mxSetAddress_NT : BOOL
VAR_INPUT
	xLSSAllowed		: BOOL;
END_VAR
VAR
	xOK 			: BOOL;
	wError 			: WORD;
	tmp 			: ARRAY [1..9] OF BYTE;
END_VAR
VAR_IN_OUT
	xStart : BOOL;
END_VAR
VAR CONSTANT
	bMaxConnectionAttempts : BYTE := 5;
END_VAR
mxSetAddress_NT := FALSE;
tonReadDelay(PT := T#50MS);

CASE bLSS_State OF 
	bSendSetAddress:
		IF bConnectionAttempts < bMaxConnectionAttempts THEN
			bConnectionAttempts := bConnectionAttempts + 1;
			CmpCanConverterWriteImage(
					wCanId 	:= 16#600+bTheAddress,
					byLen	:= 8,

					byByte0 := 16#40,
					byByte1 := 16#41,
					byByte2 := 16#60,
					byByte3 := 0,
					byByte4 := 0,
					byByte5	:= 0,
					byByte6	:= 0,
					byByte7	:= 0,
					bRemoteReq := FALSE
					);
			bLSS_State := bCheckSetAddress;
		ELSE
			bConnectionAttempts := 0;
			bLSS_State 			:= bSendDefaultAddress;
		END_IF
	
	bCheckSetAddress : 
		CmpCanConverterReadImage(wCanId := 16#580+bTheAddress,pbyMsgBfr:=ADR(tmp));
		IF tmp[1] = 16#4B AND tmp[2] = 16#41 AND tmp[3] = 16#60 THEN
			bConnectionAttempts := 0;
			bLSS_State 			:= bAddressSet;
		ELSE
			bLSS_State 			:= bSendSetAddress;
		END_IF
		
	
	bSendDefaultAddress:
		IF bConnectionAttempts < bMaxConnectionAttempts THEN
			bConnectionAttempts := bConnectionAttempts + 1;
			CmpCanConverterWriteImage(
					wCanId 	:= 16#67F,
					byLen	:= 8,

					byByte0 := 16#40,
					byByte1 := 16#41,
					byByte2 := 16#60,
					byByte3 := 0,
					byByte4 := 0,
					byByte5	:= 0,
					byByte6	:= 0,
					byByte7	:= 0,
					bRemoteReq := FALSE
					);
			bLSS_State 			:= bCheckDefaultAddress;
		ELSE
			bConnectionAttempts := 0;
			IF xLSSAllowed THEN
				bLSS_State 			:= bLSSConfig;
			ELSE
				bLSS_State 			:= bSendSetAddress;
			END_IF	
		END_IF
	
	bCheckDefaultAddress:
		CmpCanConverterReadImage(wCanId := 16#5FF,pbyMsgBfr:=ADR(tmp));
		IF tmp[1] = 16#4B AND tmp[2] = 16#41 AND tmp[3] = 16#60 THEN
			bCurrentAddress := 16#7F;
			bLSS_State 		:= bWriteAddress;
		ELSE
			bLSS_State 		:= bSendDefaultAddress;
		END_IF
	
	bLSSConfig:
		CmpCanConverterWriteImage(
						wCanId 	:= 16#7E5,
						byLen	:= 8,
						byByte0 := 16#04,
						byByte1 := 16#01,
						byByte2 := 0,
						byByte3 := 0,
						byByte4 := 0,
						byByte5	:= 0,
						byByte6	:= 0,
						byByte7	:= 0,
						bRemoteReq := FALSE
						);
		bLSS_State := bLSSRequestAddress;
	
	bLSSRequestAddress:
		IF bConnectionAttempts < bMaxConnectionAttempts THEN
			bConnectionAttempts := bConnectionAttempts + 1;	
			CmpCanConverterWriteImage(
						wCanId 	:= 16#7E5,
						byLen	:= 8,
						byByte0 := 16#5E,
						byByte1 := 0,
						byByte2 := 0,
						byByte3 := 0,
						byByte4 := 0,
						byByte5	:= 0,
						byByte6	:= 0,
						byByte7	:= 0,
						bRemoteReq := FALSE
						);
				bLSS_State := bLSSReadAddress;
		ELSE
			bConnectionAttempts := 0;
			bLSS_State 			:= bSendSetAddress;
		END_IF
	
	bLSSReadAddress:
		CmpCanConverterReadImage(wCanId := 16#7E4,pbyMsgBfr:=ADR(tmp));
		IF tmp[1] = 16#5E THEN
			bCurrentAddress := tmp[2];
			bLSS_State := bLSSWait;
		ELSE 
			bLSS_State := bLSSRequestAddress;
		END_IF
		
	bLSSWait:
		CmpCanConverterWriteImage(
						wCanId 	:= 16#7E5,
						byLen	:= 8,
						byByte0 := 16#04,
						byByte1 := 0,
						byByte2 := 0,
						byByte3 := 0,
						byByte4 := 0,
						byByte5	:= 0,
						byByte6	:= 0,
						byByte7	:= 0,
						bRemoteReq := FALSE
						);
		bLSS_State := bWriteAddress;
	
		
	bWriteAddress :
		CmpCanConverterWriteImage(
						wCanId 	:= 16#600+bCurrentAddress,
						byLen	:= 8,
						byByte0 := 16#2F,
						byByte1 := 16#09,
						byByte2 := 16#20,
						byByte3 := 16#00,
						byByte4 := bTheAddress,
						byByte5	:= 0,
						byByte6	:= 0,
						byByte7	:= 0,
						bRemoteReq := FALSE
						);
		bLSS_State := bSaveAddress;
		
	bSaveAddress:
				CmpCanConverterWriteImage(
						wCanId 	:= 16#600+bCurrentAddress,
						byLen	:= 8,
						byByte0 := 16#23,
						byByte1 := 16#10,
						byByte2 := 16#10,
						byByte3 := 16#0A,
						byByte4 := 16#73,
						byByte5	:= 16#61,
						byByte6	:= 16#76,
						byByte7	:= 16#65,
						bRemoteReq := FALSE
						);
		bLSS_State := bReset;
	

	bReset:
		fbNMTCommands.mxInit(bAddress := bCurrentAddress);
		fbNMTCommands.mxResetNode();
		bLSS_State := bAddressSet;
	
	bAddressSet:
		fbNMTCommands.mxInit(bAddress := bTheAddress);
		xStart 			:= TRUE;
		mxSetAddress_NT 	:= TRUE;
		bLSS_State 		:= bSendSetAddress;
		
ELSE
		bLSS_State := bSendSetAddress;
END_CASE
END_METHOD

METHOD mxResetAddress : BOOL
VAR_INPUT
END_VAR
VAR
	xOK 	: BOOL;
	wError 	: WORD;
	tmp 	: ARRAY [1..9] OF BYTE;
END_VAR
VAR_IN_OUT
	xStart : BOOL;
END_VAR
mxResetAddress := FALSE;

CASE bLSS_State OF 
	bResetAddress :
		CmpCanConverterWriteImage(
						wCanId 	:= 16#600+bTheAddress,
						byLen	:= 8,
						byByte0 := 16#2F,
						byByte1 := 16#09,
						byByte2 := 16#20,
						byByte3 := 16#00,
						byByte4 := 16#7F,
						byByte5	:= 0,
						byByte6	:= 0,
						byByte7	:= 0,
						bRemoteReq := FALSE
						);
		bLSS_State := bSaveAddress;
		
	bSaveAddress:
				CmpCanConverterWriteImage(
						wCanId 	:= 16#600+bTheAddress,
						byLen	:= 8,
						byByte0 := 16#23,
						byByte1 := 16#10,
						byByte2 := 16#10,
						byByte3 := 16#0A,
						byByte4 := 16#73,
						byByte5	:= 16#61,
						byByte6	:= 16#76,
						byByte7	:= 16#65,
						bRemoteReq := FALSE
						);
		bLSS_State := bReset;
	

	bReset:
		fbNMTCommands.mxResetNode();
		xStart 	:= TRUE;
		mxResetAddress 	:= TRUE;
		bLSS_State := bSendSetAddress;
ELSE
		bLSS_State := bResetAddress;
END_CASE
END_METHOD

END_FUNCTION_BLOCK

// CoolPower/PDO Topic/Tx/fbtCoolPower_CW
FUNCTION_BLOCK fbtCoolPower_CW EXTENDS fbtPDO_Word 
VAR_INPUT
END_VAR
VAR_OUTPUT
END_VAR
VAR
END_VAR

PROPERTY prpx_1_EnableVoltage : BOOL
SET
wData.1:=prpx_1_EnableVoltage;
END_SET
END_PROPERTY

PROPERTY prpx_3_EnableOperation : BOOL
SET
wData.3:=prpx_3_EnableOperation;
END_SET
END_PROPERTY

PROPERTY prpx_0_SwitchOn : BOOL
SET
wData.0:=prpx_0_SwitchOn;
END_SET
END_PROPERTY

PROPERTY prpx_4_OMS1 : BOOL
SET
wData.4:=prpx_4_OMS1;
END_SET
END_PROPERTY

PROPERTY prpx_7_FaultReset : BOOL
SET
wData.7:=prpx_7_FaultReset;
END_SET
END_PROPERTY

PROPERTY prpx_2_NoQuickStop : BOOL
SET
wData.2:=prpx_2_NoQuickStop;
END_SET
END_PROPERTY

PROPERTY prpx_8_Halt : BOOL
SET
wData.8:=prpx_8_Halt;
END_SET
END_PROPERTY

PROPERTY prpx_5_OMS2 : BOOL
SET
wData.5:=prpx_5_OMS2;
END_SET
END_PROPERTY

PROPERTY prpx_6_OMS3 : BOOL
SET
wData.6:=prpx_6_OMS3;
END_SET
END_PROPERTY

PROPERTY prpx_9_OMS4 : BOOL
SET
wData.9:=prpx_9_OMS4;
END_SET
END_PROPERTY

END_FUNCTION_BLOCK

// CoolPower/PDO Topic/Tx/fbtCoolPower_OperationMode
FUNCTION_BLOCK fbtCoolPower_OperationMode EXTENDS fbtPDO_Byte
VAR_INPUT
END_VAR
VAR_OUTPUT
END_VAR
VAR
//	bMode : BYTE := 1;
END_VAR

PROPERTY prpbOperationMode : BYTE
SET
bData := prpbOperationMode;
END_SET
END_PROPERTY

END_FUNCTION_BLOCK

// CoolPower/PDO Topic/Tx/fbtCoolPower_TargetVelocity
FUNCTION_BLOCK fbtCoolPower_TargetVelocity EXTENDS fbtPDO_DWORD
VAR_INPUT
END_VAR
VAR_OUTPUT
END_VAR
VAR
//	dwPosition : DWORD;
END_VAR

PROPERTY prpdwVelocity : DWORD
SET
dwData := prpdwVelocity;
END_SET
END_PROPERTY

END_FUNCTION_BLOCK

// CoolPower/PDO Topic/Tx/fbtCoolPower_TargetPosition
FUNCTION_BLOCK fbtCoolPower_TargetPosition EXTENDS fbtPDO_DWORD
VAR_INPUT
END_VAR
VAR_OUTPUT
END_VAR
VAR
//	dwPosition : DWORD;
END_VAR

PROPERTY prpdwPosition : DWORD
SET
dwData := prpdwPosition;
END_SET
END_PROPERTY

END_FUNCTION_BLOCK

// CoolPower/PDO Topic/Tx/fbtCoolPower_DriveSubMode
FUNCTION_BLOCK fbtCoolPower_DriveSubMode EXTENDS fbtPDO_DWord
VAR_INPUT
END_VAR
VAR_OUTPUT
END_VAR
VAR
END_VAR

PROPERTY prpx_0_ClosedLoop : BOOL
SET
dwData.0 := prpx_0_ClosedLoop;
END_SET
END_PROPERTY

PROPERTY prpx_1_VoS : BOOL
SET
dwData.1 := prpx_1_VoS;
END_SET
END_PROPERTY

PROPERTY prpx_2_Brake : BOOL
SET
dwData.2 := prpx_2_Brake;
END_SET
END_PROPERTY

PROPERTY prpx_3_CurrentReduction : BOOL
SET
dwData.3 := prpx_3_CurrentReduction;
END_SET
END_PROPERTY

PROPERTY prpx_5_Torque : BOOL
SET
dwData.5 := prpx_5_Torque;
END_SET
END_PROPERTY

PROPERTY prpx_6_BLDC : BOOL
SET
dwData.6 := prpx_6_BLDC;
END_SET
END_PROPERTY

END_FUNCTION_BLOCK

// CoolPower/PDO Topic/Tx/fbtCoolPower_ProfileVelocity
FUNCTION_BLOCK fbtCoolPower_ProfileVelocity EXTENDS fbtPDO_DWord
VAR_INPUT
END_VAR
VAR_OUTPUT
END_VAR
VAR
END_VAR

PROPERTY prpdwVelocity : DWORD
SET
dwData := prpdwVelocity;
END_SET
END_PROPERTY

END_FUNCTION_BLOCK

// CoolPower/PDO Topic/Rx/fbtCoolPower_ActualOperationMode
FUNCTION_BLOCK fbtCoolPower_ActualOperationMode EXTENDS fbtPDO_Byte
VAR_INPUT
END_VAR
VAR_OUTPUT
END_VAR
VAR
//	bMode : BYTE := 1;
END_VAR

PROPERTY prpbOperationMode : BYTE
GET
prpbOperationMode := bData;
END_GET
END_PROPERTY

END_FUNCTION_BLOCK

// CoolPower/PDO Topic/Rx/fbtCoolPower_ActualVelocity
FUNCTION_BLOCK fbtCoolPower_ActualVelocity EXTENDS fbtPDO_DWORD
VAR_INPUT
END_VAR
VAR_OUTPUT
END_VAR
VAR
//	dwPosition : DWORD;
END_VAR

PROPERTY prpdwVelocity : DWORD
GET
prpdwVelocity:=dwData;
END_GET
END_PROPERTY

END_FUNCTION_BLOCK

// CoolPower/PDO Topic/Rx/fbtCoolPower_ActualPosition
FUNCTION_BLOCK fbtCoolPower_ActualPosition EXTENDS fbtPDO_DWORD
VAR_INPUT
END_VAR
VAR_OUTPUT
END_VAR
VAR
//	dwPosition : DWORD;
END_VAR

PROPERTY prpdwPosition : DWORD
GET
prpdwPosition:=dwData;
END_GET
END_PROPERTY

END_FUNCTION_BLOCK

// CoolPower/PDO Topic/Rx/fbtCoolPower_SW
FUNCTION_BLOCK fbtCoolPower_SW EXTENDS fbtPDO_Word 
VAR_INPUT
END_VAR
VAR_OUTPUT
END_VAR
VAR
END_VAR

PROPERTY prpx_2_OperationEnabled : BOOL
GET
prpx_2_OperationEnabled:=wData.2;
END_GET
END_PROPERTY

PROPERTY prpx_0_ReadyToSwitchOn : BOOL
GET
prpx_0_ReadyToSwitchOn:=wData.0;
END_GET
END_PROPERTY

PROPERTY prpx_5_QuickStop : BOOL
GET
prpx_5_QuickStop:=wData.5;
END_GET
END_PROPERTY

PROPERTY prpx_9_Remote : BOOL
GET
prpx_9_Remote:=wData.9;
END_GET
END_PROPERTY

PROPERTY prpx_4_VoltageEnabled : BOOL
GET
prpx_4_VoltageEnabled:=wData.4;
END_GET
END_PROPERTY

PROPERTY prpx_6_SwitchOnDisabled : BOOL
GET
prpx_6_SwitchOnDisabled:=wData.6;
END_GET
END_PROPERTY

PROPERTY prpx_12_OMS1 : BOOL
GET
prpx_12_OMS1:=wData.12;
END_GET
END_PROPERTY

PROPERTY prpx_1_SwitchedOn : BOOL
GET
prpx_1_SwitchedOn:=wData.1;
END_GET
END_PROPERTY

PROPERTY prpx_7_Warning : BOOL
GET
prpx_7_Warning:=wData.7;
END_GET
END_PROPERTY

PROPERTY prpx_10_TargetReached : BOOL
GET
prpx_10_TargetReached:=wData.10;
END_GET
END_PROPERTY

PROPERTY prpx_3_Fault : BOOL
GET
prpx_3_Fault:=wData.3;
END_GET
END_PROPERTY

METHOD mbState : BYTE
VAR_INPUT
END_VAR
VAR
	wTmp : WORD;
END_VAR
wTmp := wData AND 16#000F;
CASE wTmp OF
0 : IF wData.6 THEN // wSW.prpx_6_SwitchOnDisabled 
		mbState := DS302_States.bSwitchOnDisabled;
	ELSE
		mbState := DS302_States.bNotReadyToSwitchOn;
	END_IF

1 : IF wData.5=1 AND wData.6=0 THEN
		mbState:= DS302_States.bReadyToSwitchOn;	
	ELSE
		mbState:=DS302_States.bUnknown_Error;
	END_IF

3 : IF wData.5=1 AND wData.6=0 THEN
		mbState:= DS302_States.bSwitchedOn;	
	ELSE
		mbState:=DS302_States.bUnknown_Error;
	END_IF

7 : IF wData.5=1 AND wData.6=0 THEN
		mbState:= DS302_States.bOperationEnabled;	
	ELSIF wData.5=0 AND wData.6=0 THEN
		mbState:= DS302_States.bQuickStopActive;	
	ELSE
		mbState:=DS302_States.bUnknown_Error;
	END_IF

8 : IF wData.6=0 THEN
		mbState:= DS302_States.bFault;	
	ELSE
		mbState:=DS302_States.bUnknown_Error;
	END_IF
		
16#F : IF wData.6=0 THEN
		mbState:= DS302_States.bFaultReactionActive;	
	ELSE
		mbState:=DS302_States.bUnknown_Error;
	END_IF
ELSE // case
			mbState:=DS302_States.bUnknown_Error;
END_CASE
END_METHOD

PROPERTY prpx_8_Synchronized : BOOL
GET
prpx_8_Synchronized:=wData.8;
END_GET
END_PROPERTY

PROPERTY prpx_11_InternalLimitActive : BOOL
GET
prpx_11_InternalLimitActive := wData.11;
END_GET
END_PROPERTY

PROPERTY prpx_13_OMS2 : BOOL
GET
prpx_13_OMS2:=wData.13;
END_GET
END_PROPERTY

PROPERTY prpx_15_ClosedLoop : BOOL
GET
prpx_15_ClosedLoop:=wData.15;
END_GET
END_PROPERTY

END_FUNCTION_BLOCK

// CoolPower/PDO Topic/Tx/fbtCoolPower_DigitalOutputs
FUNCTION_BLOCK fbtCoolPower_DigitalOutputs EXTENDS fbtPDO_DWORD
VAR_INPUT
END_VAR
VAR_OUTPUT
END_VAR
VAR
//	dwPosition : DWORD;
END_VAR

METHOD mxSetOutput : BOOL
VAR_INPUT
	xOutput : BOOL;
	bIndex	: BYTE;
END_VAR
VAR
	tmp		: DWORD;
END_VAR
//Create Mask
tmp.0 	:= TRUE;
tmp 	:= SHL(tmp, bIndex);

//Set or Reset bit
IF xOutput THEN
	dwData  := dwData OR tmp; 
ELSE
	tmp 	:= NOT tmp;
	dwData  := dwData AND tmp;
END_IF

mxSetOutput := TRUE;
END_METHOD

END_FUNCTION_BLOCK

// CoolPower/PDO Topic/Rx/fbtCoolPower_DigitalInputs
FUNCTION_BLOCK fbtCoolPower_DigitalInputs EXTENDS fbtPDO_DWORD
VAR_INPUT
END_VAR
VAR_OUTPUT
END_VAR
VAR
//	dwPosition : DWORD;
END_VAR

METHOD mxGetInput : BOOL
VAR_INPUT
	bIndex	: BYTE;
END_VAR
VAR_OUTPUT
	xInput	: BOOL;
END_VAR
VAR
	tmp 	: DWORD;
END_VAR
//Shift Request to Bit 0
tmp 	:= dwData;
tmp 	:= SHR(tmp,bIndex);

//Read Input
xInput 	:= tmp.0;

mxGetInput := TRUE;
END_METHOD

END_FUNCTION_BLOCK

// CoolPower/PDO Topic/Rx/fbtCoolPower_MaxMotorSpeed
FUNCTION_BLOCK fbtCoolPower_MaxMotorSpeed EXTENDS fbtPDO_DWORD
VAR_INPUT
END_VAR
VAR_OUTPUT
END_VAR
VAR
//	dwPosition : DWORD;
END_VAR

PROPERTY prpdwMaxSpeed : DWORD
GET
prpdwMaxSpeed:=dwData;
END_GET
END_PROPERTY

END_FUNCTION_BLOCK

// CoolPower/PDO Topic/Rx/fbtCoolPower_RunningHours
FUNCTION_BLOCK fbtCoolPower_RunningHours EXTENDS fbtPDO_DWORD
VAR_INPUT
END_VAR
VAR_OUTPUT
END_VAR
VAR
//	dwPosition : DWORD;
END_VAR

PROPERTY prpdwRunningHours : DWORD
GET
prpdwRunningHours:=dwData;
END_GET
END_PROPERTY

END_FUNCTION_BLOCK

// CoolPower/PDO Topic/Rx/fbtCoolPower_SerialNumber_1_6
FUNCTION_BLOCK fbtCoolPower_SerialNumber_1_6 EXTENDS fbtPDO_DWORD
VAR_INPUT
END_VAR
VAR_OUTPUT
END_VAR
VAR
//	dwPosition : DWORD;
END_VAR

PROPERTY prpdwSerial_1_6 : DWORD
GET
prpdwSerial_1_6:=dwData;
END_GET
END_PROPERTY

END_FUNCTION_BLOCK

// CoolPower/PDO Topic/Rx/fbtCoolPower_SerialNumber_7_11
FUNCTION_BLOCK fbtCoolPower_SerialNumber_7_11 EXTENDS fbtPDO_DWORD
VAR_INPUT
END_VAR
VAR_OUTPUT
END_VAR
VAR
//	dwPosition : DWORD;
END_VAR

PROPERTY prpdwSerial_7_11 : DWORD
GET
prpdwSerial_7_11:=dwData;
END_GET
END_PROPERTY

END_FUNCTION_BLOCK

// CoolPower/fbtCoolPower_NanoTec
FUNCTION_BLOCK fbtCoolPower_NanoTec
VAR_INPUT
END_VAR
VAR_OUTPUT
END_VAR
VAR
	bMyCANAddress			: BYTE;
	xStartLocal				: BOOL;
	
	fbCANOpen 				: fbtCANOpenDriver_CoolPower;
	CoolPower_SN_1_6		: fbtSDOCouple;
 	CoolPower_SN_7_11		: fbtSDOCouple;
 	CoolPower_RunningHours	: fbtSDOCouple;
	CoolPower_TotalHours	: fbtSDOCouple;
 	CoolPower_MaxSpeed		: fbtSDOCouple;
	CoolPower_HourReset		: fbtSDOCouple;
	CoolPower_Model			: fbtSDOCouple;
	
	CoolPower_CW 			: fbtCoolPower_CW;
	CoolPower_OpMode 		: fbtCoolPower_OperationMode;
	CoolPower_TargetVel		: fbtCoolPower_TargetVelocity;
	CoolPower_DO			: fbtCoolPower_DigitalOutputs;

	CoolPower_SW			: fbtCoolPower_SW;
	CoolPower_ActualOpMode	: fbtCoolPower_ActualOperationMode;
	CoolPower_ActualVel		: fbtCoolPower_ActualVelocity;
	CoolPower_DI			: fbtCoolPower_DigitalInputs;	
	
	CoolPower_List			: fbtSDO_Series_CoolPower;

	Tp_CommandTimeOut		: TP;
	xStartTimeOut			: BOOL;
	bDriveState				: BYTE;
	bReadOutState			: BYTE;
	bConfigurationState		: BYTE;
	bResetState				: BYTE;
	sdoWrite				: SingleFullSDO;
END_VAR
VAR CONSTANT
	bNewReadout				: BYTE := 0;
	bSerialPartial			: BYTE := 1;
	bSerialFinished			: BYTE := 2;
	bRunningHours			: BYTE := 3;
	bTotalHours				: BYTE := 4;
	bMaxSpeed				: BYTE := 5;
	bModel					: BYTE := 6;
	bReadOutDone			: BYTE := 7;
	bLSS					: BYTE := 0;
	bSetPreOp				: BYTE := 1;
	bDeactivatePDO			: BYTE := 2;
	bCreateMapping			: BYTE := 3;
	bActivatePDO			: BYTE := 4;
	bCheckReset 			: BYTE := 0;
	bSendPulse 				: BYTE := 1;
	bCheckCounter			: BYTE := 2;
	bResetPulse				: BYTE := 3;	
END_VAR

PROPERTY prpbOperationMode : BYTE
GET
prpbOperationMode := CoolPower_ActualOpMode.prpbOperationMode;
END_GET
SET
CoolPower_OpMode.prpbOperationMode := prpbOperationMode;
END_SET
END_PROPERTY

PROPERTY prpdwMaxSpeed : DWORD
GET
VAR
	 i 			: INT;
	 tmpItem 	: DWORD;
END_VAR
prpdwMaxSpeed := 0;
FOR i := 4 TO 7 DO
	tmpItem := 0;
	tmpItem := CoolPower_MaxSpeed.prppMessageIn^.data[i];
	tmpItem := SHL(tmpItem,8*(i - 4));
	prpdwMaxSpeed := prpdwMaxSpeed OR tmpItem;
END_FOR
END_GET
END_PROPERTY

PROPERTY prpdwRunningHours : DWORD
GET
VAR
	 i 			: INT;
	 tmpItem	: DWORD;
END_VAR
prpdwRunningHours := 0;
FOR i := 4 TO 7 DO
	tmpItem := 0;
	tmpItem := CoolPower_RunningHours.prppMessageIn^.data[i];
	tmpItem := SHL(tmpItem,8*(i - 4));
	prpdwRunningHours := prpdwRunningHours OR tmpItem;
END_FOR
END_GET
END_PROPERTY

PROPERTY prpdwSpeed : DWORD
GET
prpdwSpeed := CoolPower_ActualVel.prpdwVelocity;
END_GET
SET
CoolPower_TargetVel.prpdwVelocity := prpdwSpeed;
END_SET
END_PROPERTY

PROPERTY prpulSerialNumber : ULINT
GET
VAR
	 i : INT;
	 dwTempHigh : DWORD;
	 dwTempLow	: DWORD;
	 tmpItem	: DWORD;
END_VAR
dwTempHigh := 0;
FOR i := 4 TO 7 DO
	tmpItem := 0;
	tmpItem := CoolPower_SN_1_6.prppMessageIn^.data[i];
	tmpItem := SHL(tmpItem,8*(i - 4));
	dwTempHigh := dwTempHigh OR tmpItem;
END_FOR
dwTempLow := 0;
FOR i := 4 TO 7 DO
	tmpItem := 0;
	tmpItem := CoolPower_SN_7_11.prppMessageIn^.data[i];
	tmpItem := SHL(tmpItem,8*(i - 4));
	dwTempLow := dwTempLow OR tmpItem;
END_FOR

prpulSerialNumber := DWORD_TO_ULINT(dwTempHigh) * 100000 + DWORD_TO_ULINT(dwTempLow);
END_GET
END_PROPERTY

PROPERTY prpxHalt : BOOL
SET
CoolPower_CW.prpx_8_Halt := prpxHalt;
END_SET
END_PROPERTY

PROPERTY prpxIsOperational : BOOL
GET
prpxIsOperational := fbCANOpen.prpxIsOperational;
END_GET
END_PROPERTY

PROPERTY prpbModel : BYTE
GET
VAR
	 i 			: INT;
	 tmpItem 	: DWORD;
END_VAR
prpbModel := CoolPower_Model.prppMessageIn^.data[4];
END_GET
END_PROPERTY

PROPERTY prpdwTotalHours : DWORD
GET
VAR
	 i 			: INT;
	 tmpItem	: DWORD;
END_VAR
prpdwTotalHours := 0;
FOR i := 4 TO 7 DO
	tmpItem := 0;
	tmpItem := CoolPower_TotalHours.prppMessageIn^.data[i];
	tmpItem := SHL(tmpItem,8*(i - 4));
	prpdwTotalHours := prpdwTotalHours OR tmpItem;
END_FOR
END_GET
END_PROPERTY

METHOD mxDisable : BOOL
VAR_INPUT
END_VAR
VAR_IN_OUT
	xStart : BOOL;
END_VAR
VAR_OUTPUT
	xOK 	: BOOL;
	wError 	: WORD;
END_VAR
mxDisable:=FALSE;

IF xStart THEN
	xStart:=FALSE;
	xStartTimeOut:=TRUE;
	Tp_CommandTimeOut(IN:=FALSE,PT:=T#4S); 
	wError:=0;
END_IF

Tp_CommandTimeOut(IN:=xStartTimeOut,PT:=T#4S); // time to be defined
IF NOT Tp_CommandTimeOut.Q THEN
	wError:=1;
	mxDisable:=TRUE;
	RETURN;
END_IF

CASE bDriveState OF
	DS302_States.bNoInfo 	 		 :
		bDriveState	:= CoolPower_SW.mbState();
	
	DS302_States.bNotReadyToSwitchOn 	: 
		bDriveState	:= CoolPower_SW.mbState();
		mxDisable 	:= FALSE;
		
	DS302_States.bSwitchOnDisabled 	: 
		bDriveState	:= CoolPower_SW.mbState();
		mxDisable 	:= TRUE;

	DS302_States.bReadyToSwitchOn,
	DS302_States.bSwitchedOn,
	DS302_States.bOperationEnabled,
	DS302_States.bQuickStopActive:
		CoolPower_TargetVel.prpdwVelocity := 0;
		CoolPower_CW.mxClear();
		bDriveState			:= CoolPower_SW.mbState();
	
	DS302_States.bFaultReactionActive,
	DS302_States.bFault,
	DS302_States.bUnknown_Error:
		CoolPower_TargetVel.prpdwVelocity := 0;
		CoolPower_CW.mxClear();
		mxDisable 	:= TRUE;	
END_CASE
END_METHOD

METHOD mxEnable : BOOL
VAR_INPUT
END_VAR
VAR_IN_OUT
	xStart : BOOL;
END_VAR
VAR_OUTPUT
	xOK 	: BOOL;
	wError 	: WORD;
END_VAR
mxEnable	:=FALSE;
wError		:=0;

IF xStart THEN
	xStart			:=FALSE;
	xStartTimeOut	:=TRUE;
	bDriveState		:=CoolPower_SW.mbState();
	Tp_CommandTimeOut(IN:=FALSE,PT:=T#4S); 
END_IF

// Startup time-out timer, triggers if it takes too long to get this startup => problem
Tp_CommandTimeOut(IN:=xStartTimeOut,PT:=T#6S); // time to be defined
IF NOT Tp_CommandTimeOut.Q THEN
	wError	:=1;
	mxEnable:=TRUE;
END_IF
xStartTimeOut:=FALSE;
// CANOpen drive states
CASE bDriveState OF
	DS302_States.bNoInfo 	 		 :
		bDriveState:=CoolPower_SW.mbState();

	DS302_States.bNotReadyToSwitchOn 	: 
		bDriveState:=CoolPower_SW.mbState();

	DS302_States.bSwitchOnDisabled  	: // transition 2 -> Ready Switch On
		// set appropriate bits to continue
		CoolPower_CW.prpx_0_SwitchOn		:= FALSE;
		CoolPower_CW.prpx_1_EnableVoltage	:= TRUE;
		CoolPower_CW.prpx_2_NoQuickStop		:= TRUE;
		CoolPower_CW.prpx_3_EnableOperation	:= FALSE;
		CoolPower_CW.prpx_7_FaultReset 		:= FALSE;
		bDriveState:=CoolPower_SW.mbState();
		
	DS302_States.bReadyToSwitchOn   	: // transition 3 -> Switched On
		// set appropriate bits to continue
		CoolPower_CW.prpx_0_SwitchOn		:=TRUE;
		CoolPower_CW.prpx_1_EnableVoltage	:=TRUE;
		CoolPower_CW.prpx_2_NoQuickStop		:=TRUE;
		CoolPower_CW.prpx_3_EnableOperation	:=FALSE;
		bDriveState:=CoolPower_SW.mbState();

	DS302_States.bSwitchedOn 		  	: // transition 4 -> Operation Enabled
		// set appropriate bits to continue
		CoolPower_CW.prpx_0_SwitchOn		:=TRUE;
		CoolPower_CW.prpx_1_EnableVoltage	:=TRUE;
		CoolPower_CW.prpx_2_NoQuickStop		:=TRUE;
		CoolPower_CW.prpx_3_EnableOperation	:=TRUE;
		bDriveState:=CoolPower_SW.mbState();
		
	DS302_States.bOperationEnabled  	: // stay at operation enabled
		CoolPower_CW.prpx_0_SwitchOn		:=TRUE;
		CoolPower_CW.prpx_1_EnableVoltage	:=TRUE;
		CoolPower_CW.prpx_2_NoQuickStop		:=TRUE;
		CoolPower_CW.prpx_3_EnableOperation	:=TRUE;
		mxEnable :=TRUE; 			// startup ok
		bConfigurationState 				:= bSetPreOp;
		
	DS302_States.bQuickStopActive  	: // transition 16 -> Operation Enabled 
		// start from QuickStop with speed:=0;
		CoolPower_CW.prpx_0_SwitchOn		:=TRUE;
		CoolPower_CW.prpx_1_EnableVoltage	:=TRUE;
		CoolPower_CW.prpx_2_NoQuickStop		:=TRUE;
		CoolPower_CW.prpx_3_EnableOperation	:=TRUE;
		bDriveState:=CoolPower_SW.mbState();
		
	DS302_States.bFault, DS302_States.bFaultReactionActive, DS302_States.bUnknown_Error :
		CoolPower_CW.mxClear();
		CoolPower_CW.prpx_7_FaultReset := TRUE;
		wError		:=2;
		mxEnable	:=TRUE;
END_CASE;
END_METHOD

METHOD mxInit : BOOL
VAR_INPUT
	bCANAddress : BYTE;
END_VAR
bMyCANAddress := bCANAddress;

fbCANOpen.mxInit(	bCANAddress 			:= bCANAddress);
					

fbCANOpen.mxClearPDOConfiguration();

fbCANOpen.mxAddTxPDOTopic(1, CoolPower_CW);
fbCANOpen.mxAddTxPDOTopic(1, CoolPower_OpMode);
fbCANOpen.mxAddTxPDOTopic(1, CoolPower_TargetVel);

fbCANOpen.mxAddTxPDOTopic(2, CoolPower_DO);

fbCANOpen.mxAddRxPDOTopic(1, CoolPower_SW			, TRUE, 10000); 
fbCANOpen.mxAddRxPDOTopic(1, CoolPower_ActualOpMode	, TRUE, 10000); 
fbCANOpen.mxAddRxPDOTopic(1, CoolPower_ActualVel	, TRUE, 10000); 

fbCANOpen.mxAddRxPDOTopic(2, CoolPower_DI			, TRUE, 10000);

bConfigurationState := bLSS;
END_METHOD

METHOD mxRun : BOOL
VAR_INPUT
END_VAR
VAR
	xOk		: BOOL;
	wError	: WORD;
END_VAR
fbCanOpen.mxRun();
END_METHOD

METHOD mxReadOut : BOOL
VAR_INPUT
END_VAR
VAR_IN_OUT
	xStart : BOOL;
END_VAR
VAR_OUTPUT
	xOK		: BOOL;
	xReady 	: BOOL;
	wError 	: WORD;
END_VAR
mxReadOut := FALSE;
IF xStart THEN
	bReadOutState := bNewReadout;
	xStartLocal := TRUE;
	xStart 		:= FALSE;
END_IF

CASE bReadOutState OF
	bNewReadout: 
		IF xStartLocal THEN
			IF prpulSerialNumber <> 0 THEN
				CoolPower_RunningHours.mxMakeRead_Idx(
													bMyCANAddress,
													GVL_NanoTecAddresses.RunningHours_Index,		
													GVL_NanoTecAddresses.RunningHours_Subindex
												);
				bReadOutState := bRunningHours;
			ELSE
				CoolPower_SN_1_6.mxMakeRead_Idx(		
												bMyCANAddress,
												GVL_NanoTecAddresses.SerialNumber1_6_Index,	
												GVL_NanoTecAddresses.SerialNumber1_6_Subindex
											);
				bReadOutState := bSerialPartial;
			END_IF
		END_IF
	
	bSerialPartial:
		IF fbCANOpen.prpitfCANOpen_SDO.mxSDORead_Safe(itfSDOCouple := CoolPower_SN_1_6,xStart := xStartLocal, xOK => xOK) THEN
			xStartLocal := TRUE;
			IF xOK THEN
				CoolPower_SN_7_11.mxMakeRead_Idx(
												bMyCANAddress,
												GVL_NanoTecAddresses.SerialNumber7_11_Index,
												GVL_NanoTecAddresses.SerialNumber7_11_Subindex
											);
				bReadOutState := bSerialFinished;
			END_IF					
		END_IF
		
	bSerialFinished:
		IF fbCANOpen.prpitfCANOpen_SDO.mxSDORead_Safe(itfSDOCouple := CoolPower_SN_7_11,xStart :=  xStartLocal, xOK => xOK) THEN
			xStartLocal := TRUE;
			IF xOK THEN
				CoolPower_RunningHours.mxMakeRead_Idx(	
													bMyCANAddress,
													GVL_NanoTecAddresses.RunningHours_Index,	
													GVL_NanoTecAddresses.RunningHours_Subindex
												);
				bReadOutState := bRunningHours;
			END_IF				
		END_IF
		
	bRunningHours:
		IF fbCANOpen.prpitfCANOpen_SDO.mxSDORead_Safe(itfSDOCouple := CoolPower_RunningHours, xStart :=  xStartLocal, xOK => xOK) THEN
			xStartLocal := TRUE;
			IF xOK THEN
				CoolPower_TotalHours.mxMakeRead_Idx(		
												bMyCANAddress,
												GVL_NanoTecAddresses.TotalHours_Index,	
												GVL_NanoTecAddresses.TotalHours_Subindex
											);
				bReadOutState := bTotalHours;				
			END_IF
		END_IF
		
	bTotalHours:
		IF fbCANOpen.prpitfCANOpen_SDO.mxSDORead_Safe(itfSDOCouple := CoolPower_TotalHours, xStart :=  xStartLocal, xOK => xOK) THEN
			xStartLocal := TRUE;
			IF xOK THEN
				CoolPower_MaxSpeed.mxMakeRead_Idx(		
												bMyCANAddress,
												GVL_NanoTecAddresses.MaxSpeed_Index,	
												GVL_NanoTecAddresses.MaxSpeed_Subindex
											);
				bReadOutState := bMaxSpeed;				
			END_IF
		END_IF
	
	
	bMaxSpeed:
		IF fbCANOpen.prpitfCANOpen_SDO.mxSDORead_Safe(itfSDOCouple := CoolPower_MaxSpeed,xStart := xStartLocal,xOK => xOK) THEN
			xStartLocal := TRUE;
			IF xOK THEN
				CoolPower_Model.mxMakeRead_Idx(		
												bMyCANAddress,
												GVL_NanoTecAddresses.Model_Index,	
												GVL_NanoTecAddresses.Model_Subindex
											);
				bReadOutState := bModel;			
			END_IF
		END_IF
		
	bModel:
		IF fbCANOpen.prpitfCANOpen_SDO.mxSDORead_Safe(itfSDOCouple := CoolPower_Model,xStart := xStartLocal,xOK => xOK) THEN
			xStartLocal := TRUE;
			IF xOK THEN	
				IF prpbModel <> 0 THEN
						bReadOutState := bReadOutDone;
					ELSE
						bReadOutState := bNewReadout;
				END_IF	
			END_IF
		END_IF

	bReadOutDone:	
		mxReadOut := TRUE;		
END_CASE
END_METHOD

METHOD mxConfigure : BOOL
VAR_INPUT
	xLSSAllowed : BOOL;
END_VAR
VAR
	xOK			: BOOL;
END_VAR
VAR_IN_OUT
	xStart		:  BOOL;
END_VAR
CASE bConfigurationState OF 
	bLSS:
		IF fbCANOpen.mxSetAddress_NT(xStart := xStart, xLSSAllowed := xLSSAllowed) THEN
			bConfigurationState := bSetPreOp;
			xStart 				:= TRUE;
		END_IF
		
	bSetPreOp: 
		IF fbCANOpen.mxConfigPrep() THEN
			bConfigurationState := 	bDeactivatePDO;
		END_IF
		
		
	bDeactivatePDO:
		CoolPower_List.prpbAddress := bMyCANAddress;
		CoolPower_List.mxInitList();
		bConfigurationState := bCreateMapping;
		
	bCreateMapping:
		IF fbCanOpen.prpitfCANOpen_SDO.mxWriteFullList(bMyCANAddress,CoolPower_List,xStart,xOk=>xOK) THEN
			IF xOK THEN
				bConfigurationState :=bActivatePDO;
				fbCANOpen.mxReset();
			END_IF
			xStart := TRUE;
		END_IF
		
	bActivatePDO:
			mxConfigure := TRUE;
END_CASE
END_METHOD

METHOD mxReset : BOOL
VAR_INPUT
END_VAR
bConfigurationState := bLSS;
fbCANOpen.mxReset();
END_METHOD

METHOD mxClean : BOOL
VAR
	xOK			: BOOL;
END_VAR
VAR_IN_OUT
	xStart		:  BOOL;
END_VAR
CASE bConfigurationState OF 
	bSetPreOp: 
		IF fbCANOpen.mxConfigPrep() THEN
			bConfigurationState := bLSS;
		END_IF
		
	bLSS:
		IF fbCANOpen.mxResetAddress(xStartLocal) THEN
			bConfigurationState := bActivatePDO;
			xStartLocal 				:= TRUE;
		END_IF
		
	bActivatePDO:
			CoolPower_SN_1_6.mxMakeRead_Idx(		
											bMyCANAddress,
											GVL_NanoTecAddresses.SerialNumber1_6_Index,	
											GVL_NanoTecAddresses.SerialNumber1_6_Subindex
										);
			CoolPower_SN_7_11.mxMakeRead_Idx(
											bMyCANAddress,
											GVL_NanoTecAddresses.SerialNumber7_11_Index,
											GVL_NanoTecAddresses.SerialNumber7_11_Subindex
										);
			CoolPower_RunningHours.mxMakeRead_Idx(	
												bMyCANAddress,
												GVL_NanoTecAddresses.RunningHours_Index,	
												GVL_NanoTecAddresses.RunningHours_Subindex
											);
			CoolPower_MaxSpeed.mxMakeRead_Idx(		
											bMyCANAddress,
											GVL_NanoTecAddresses.MaxSpeed_Index,	
											GVL_NanoTecAddresses.MaxSpeed_Subindex
										);
			mxClean 	:= TRUE;
			xStart 		:= TRUE;
			bConfigurationState := bLSS;
ELSE
		bConfigurationState := bSetPreOp;
END_CASE
END_METHOD

METHOD mxResetCounter : BOOL
VAR_INPUT
	xStartReset : BOOL;
END_VAR
VAR
	xOK : BOOL;
END_VAR
CASE bResetState OF
	bCheckReset:	
		IF xStartReset THEN
			//Create Reset Message
			sdoWrite.wIndex 			:= 16#2400;
			sdoWrite.bSubIndex 			:= 16#01;
			sdoWrite.bLgt 				:= 4;
			sdoWrite.odValue.dwValue	:= 1;
			sdoWrite.pbValue			:= 0;
			sdoWrite.wDelay 			:= 1;
			CoolPower_HourReset.mxMakeWriteFull(bAddress:= bMyCANAddress,pSDO := ADR(sdoWrite));
			
			//Setup Local Start
			xStartLocal := TRUE;
			
			//Start Reset Cycle
			bResetState := bSendPulse;
		END_IF
	
		
	bSendPulse:
		//Write Reset Message
		IF fbCanOpen.prpitfCANOpen_SDO.mxSDOWrite_Safe(CoolPower_HourReset, xStart := xStartLocal,xOK => xOK) THEN
			xStartLocal := TRUE;
			IF xOK THEN
				//Create Reading Message
				CoolPower_RunningHours.mxMakeRead_Idx(
													bMyCANAddress,
													GVL_NanoTecAddresses.RunningHours_Index,		
													GVL_NanoTecAddresses.RunningHours_Subindex
												);
				//Read Running Hours
				bResetState := bCheckCounter;
			END_IF
		END_IF
		

										
	bCheckCounter:
		IF fbCanOpen.prpitfCANOpen_SDO.mxSDORead_Safe(CoolPower_RunningHours, xStart := xStartLocal, xOK => xOK) THEN
			xStartLocal := TRUE;
			IF xOK AND_THEN prpdwRunningHours = 0 THEN
				//Create Reset Message Recall
				sdoWrite.wIndex 			:= 16#2400;
				sdoWrite.bSubIndex 			:= 16#01;
				sdoWrite.bLgt 				:= 4;
				sdoWrite.odValue.dwValue	:= 0;
				sdoWrite.pbValue			:= 0;
				sdoWrite.wDelay 			:= 1;
				CoolPower_HourReset.mxMakeWriteFull(bAddress:= bMyCANAddress,pSDO := ADR(sdoWrite));
				
				//Send Reset Message Recall
				bResetState := bResetPulse;
			END_IF
		END_IF
		
	bResetPulse:
		IF fbCanOpen.prpitfCANOpen_SDO.mxSDOWrite_Safe(CoolPower_HourReset, xStart := xStartLocal,xOK => xOK) THEN
			xStartLocal := TRUE;
			IF xOK THEN
				bResetState := bCheckReset;
				mxResetCounter := TRUE;
			END_IF
		END_IF
END_CASE
END_METHOD

END_FUNCTION_BLOCK

// CoolPower/CANOpenDriver/fbtSDO_Series_CoolPower
FUNCTION_BLOCK fbtSDO_Series_CoolPower EXTENDS fbtSDO_FullList_Base
VAR_INPUT
END_VAR
VAR_OUTPUT
END_VAR
VAR
	SDOList		: ARRAY [0..wListLength] OF SingleFullSDO;
	bAddress	: BYTE;
END_VAR
VAR CONSTANT
	wListLength	: WORD := 28;
END_VAR

METHOD mxGetSDO : BOOL
VAR_INPUT
	wNr	: WORD;
END_VAR
VAR_OUTPUT
	pTheSDO	: POINTER TO SingleFullSDO;
END_VAR
pTheSDO := ADR(SDOList[wNr]);
mxGetSDO := wNr >= 0 AND wNr <= wListLength;
END_METHOD

METHOD mxInitList : BOOL
SysMemSet(ADR(SDOList),0,SIZEOF(SDOList));

//Disable PDO's
SDOList[1].wIndex 			:= 16#1400;
SDOList[1].bSubIndex 		:= 16#01;
SDOList[1].bLgt				:= 4;
SDOList[1].odValue.dwValue	:= 16#80000200+bAddress;
SDOList[1].wDelay			:= 0;
SDOList[2].wIndex 			:= 16#1401;
SDOList[2].bSubIndex 		:= 16#01;
SDOList[2].bLgt				:= 4;
SDOList[2].odValue.dwValue	:= 16#80000300+bAddress;
SDOList[2].wDelay			:= 0;
SDOList[3].wIndex 			:= 16#1800;
SDOList[3].bSubIndex 		:= 16#01;
SDOList[3].bLgt				:= 4;
SDOList[3].odValue.dwValue	:= 16#80000180+bAddress;
SDOList[3].wDelay			:= 0;
SDOList[4].wIndex 			:= 16#1801;
SDOList[4].bSubIndex 		:= 16#01;
SDOList[4].bLgt				:= 4;
SDOList[4].odValue.dwValue	:= 16#80000280+bAddress;
SDOList[4].wDelay			:= 0;

//Set Transmission type to continuous sending
SDOList[5].wIndex 			:= 16#1800;
SDOList[5].bSubIndex 		:= 16#02;
SDOList[5].bLgt				:= 1;
SDOList[5].odValue.dwValue	:= 16#FF;
SDOList[5].wDelay			:= 0;
SDOList[6].wIndex 			:= 16#1801;
SDOList[6].bSubIndex 		:= 16#02;
SDOList[6].bLgt				:= 1;
SDOList[6].odValue.dwValue	:= 16#FF;
SDOList[6].wDelay			:= 0;
SDOList[7].wIndex 			:= 16#1800;
SDOList[7].bSubIndex 		:= 16#05;
SDOList[7].bLgt				:= 2;
SDOList[7].odValue.dwValue	:= 16#01F4;
SDOList[7].wDelay			:= 0;
SDOList[8].wIndex 			:= 16#1801;
SDOList[8].bSubIndex 		:= 16#05;
SDOList[8].bLgt				:= 2;
SDOList[8].odValue.dwValue	:= 16#01F4;
SDOList[8].wDelay			:= 0;

//Set Rx-PDO Mapping
SDOList[9].wIndex 			:= 16#1600;
SDOList[9].bSubIndex 		:= 16#00;
SDOList[9].bLgt				:= 1;
SDOList[9].odValue.dwValue	:= 16#00;
SDOList[9].wDelay			:= 0;
SDOList[10].wIndex 			:= 16#1600;
SDOList[10].bSubIndex 		:= 16#01;
SDOList[10].bLgt			:= 4;
SDOList[10].odValue.dwValue	:= 16#60400010;
SDOList[10].wDelay			:= 0;
SDOList[11].wIndex 			:= 16#1600;
SDOList[11].bSubIndex 		:= 16#02;
SDOList[11].bLgt			:= 4;
SDOList[11].odValue.dwValue	:= 16#60600008;
SDOList[11].wDelay			:= 0;
SDOList[12].wIndex 			:= 16#1600;
SDOList[12].bSubIndex 		:= 16#03;
SDOList[12].bLgt			:= 4;
SDOList[12].odValue.dwValue	:= 16#60FF0020;
SDOList[12].wDelay			:= 0;
SDOList[13].wIndex 			:= 16#1600;
SDOList[13].bSubIndex 		:= 16#00;
SDOList[13].bLgt			:= 1;
SDOList[13].odValue.dwValue	:= 16#03;
SDOList[13].wDelay			:= 0;
SDOList[14].wIndex 			:= 16#1601;
SDOList[14].bSubIndex 		:= 16#00;
SDOList[14].bLgt			:= 1;
SDOList[14].odValue.dwValue	:= 16#00;
SDOList[14].wDelay			:= 0;
SDOList[15].wIndex 			:= 16#1601;
SDOList[15].bSubIndex 		:= 16#01;
SDOList[15].bLgt			:= 4;
SDOList[15].odValue.dwValue	:= 16#60FE0120;
SDOList[15].wDelay			:= 0;
SDOList[16].wIndex 			:= 16#1601;
SDOList[16].bSubIndex 		:= 16#00;
SDOList[16].bLgt			:= 1;
SDOList[16].odValue.dwValue	:= 16#01;
SDOList[16].wDelay			:= 0;


//Set Tx-PDO Mapping
SDOList[17].wIndex 			:= 16#1A00;
SDOList[17].bSubIndex 		:= 16#00;
SDOList[17].bLgt			:= 1;
SDOList[17].odValue.dwValue	:= 16#00;
SDOList[17].wDelay			:= 0;
SDOList[18].wIndex 			:= 16#1A00;
SDOList[18].bSubIndex 		:= 16#01;
SDOList[18].bLgt			:= 4;
SDOList[18].odValue.dwValue	:= 16#60410010;
SDOList[18].wDelay			:= 0;
SDOList[19].wIndex 			:= 16#1A00;
SDOList[19].bSubIndex 		:= 16#02;
SDOList[19].bLgt			:= 4;
SDOList[19].odValue.dwValue	:= 16#60610008;
SDOList[19].wDelay			:= 0;
SDOList[20].wIndex 			:= 16#1A00;
SDOList[20].bSubIndex 		:= 16#03;
SDOList[20].bLgt			:= 4;
SDOList[20].odValue.dwValue	:= 16#606C0020;
SDOList[20].wDelay			:= 0;
SDOList[21].wIndex 			:= 16#1A00;
SDOList[21].bSubIndex 		:= 16#00;
SDOList[21].bLgt			:= 1;
SDOList[21].odValue.dwValue	:= 16#03;
SDOList[21].wDelay			:= 0;
SDOList[22].wIndex 			:= 16#1A01;
SDOList[22].bSubIndex 		:= 16#00;
SDOList[22].bLgt			:= 1;
SDOList[22].odValue.dwValue	:= 16#00;
SDOList[22].wDelay			:= 0;
SDOList[23].wIndex 			:= 16#1A01;
SDOList[23].bSubIndex 		:= 16#01;
SDOList[23].bLgt			:= 4;
SDOList[23].odValue.dwValue	:= 16#60FD0020;
SDOList[23].wDelay			:= 0;
SDOList[24].wIndex 			:= 16#1A01;
SDOList[24].bSubIndex 		:= 16#00;
SDOList[24].bLgt			:= 1;
SDOList[24].odValue.dwValue	:= 16#01;
SDOList[24].wDelay			:= 0;

//Reactivate PDO's
SDOList[25].wIndex 			:= 16#1400;
SDOList[25].bSubIndex 		:= 16#01;
SDOList[25].bLgt			:= 4;
SDOList[25].odValue.dwValue	:= 16#00000200+bAddress;
SDOList[25].wDelay			:= 0;
SDOList[26].wIndex 			:= 16#1401;
SDOList[26].bSubIndex 		:= 16#01;
SDOList[26].bLgt			:= 4;
SDOList[26].odValue.dwValue	:= 16#00000300+bAddress;
SDOList[26].wDelay			:= 0;
SDOList[27].wIndex 			:= 16#1800;
SDOList[27].bSubIndex 		:= 16#01;
SDOList[27].bLgt			:= 4;
SDOList[27].odValue.dwValue	:= 16#00000180+bAddress;
SDOList[27].wDelay			:= 0;
SDOList[28].wIndex 			:= 16#1801;
SDOList[28].bSubIndex 		:= 16#01;
SDOList[28].bLgt			:= 4;
SDOList[28].odValue.dwValue	:= 16#00000280+bAddress;
SDOList[28].wDelay			:= 0;

wPointer 	:= 0;
wNrSDO		:= wListLength;
END_METHOD

PROPERTY prpbAddress : BYTE
SET
bAddress := prpbAddress;
END_SET
END_PROPERTY

END_FUNCTION_BLOCK

// Aorta/Driver/Settings/fbtAorta_AllSettings_Tri
FUNCTION_BLOCK fbtAorta_AllSettings_Tri EXTENDS fbtSDO_FullList_Base 
VAR_INPUT
END_VAR
VAR_OUTPUT
END_VAR
VAR
	AllSettings : ARRAY[1..25] OF SingleFullSDO;
END_VAR

METHOD mxInit : BOOL
VAR_INPUT
END_VAR
VAR
	i : WORD;
	TmpItem	: ODItem;
END_VAR
i:=1;

SysMemSet(ADR(AllSettings[i]),0,SIZEOF(AllSettings[i]));

// Absolute Maximum Current
CmpODRead(ENUM_SDO_2000.Aorta,	12,	ADR(TmpItem));
AllSettings[i].wIndex:=16#2003;
AllSettings[i].bSubIndex:=0;
AllSettings[i].bLgt:=1;
AllSettings[i].odValue.bValue[1]:=TmpItem.bValue[1];//120;
// Standby Current
i:=i+1;
CmpODRead(ENUM_SDO_2000.Aorta,	12,	ADR(TmpItem));
AllSettings[i].wIndex:=16#2004;
AllSettings[i].bSubIndex:=0;
AllSettings[i].bLgt:=1;
AllSettings[i].odValue.bValue[1]:=TmpItem.bValue[2];//8;
//
// Homing
//
// Expected Homing Time Min
i:=i+1;
CmpODRead(ENUM_SDO_2000.Aorta,	13,	ADR(TmpItem));
AllSettings[i].wIndex:=16#20C0;
AllSettings[i].bSubIndex:=1;
AllSettings[i].bLgt:=4;
AllSettings[i].odValue.dwValue:=TmpItem.dwValue;//0;
// Expected Homing Time Max
i:=i+1;
CmpODRead(ENUM_SDO_2000.Aorta,	14,	ADR(TmpItem));
AllSettings[i].wIndex:=16#20C0;
AllSettings[i].bSubIndex:=2;
AllSettings[i].bLgt:=4;
AllSettings[i].odValue.dwValue:=TmpItem.dwValue;//0;
// StallGuard Threshold
i:=i+1;
CmpODRead(ENUM_SDO_2000.Aorta,	12,	ADR(TmpItem));
AllSettings[i].wIndex:=16#209E;
AllSettings[i].bSubIndex:=2;
AllSettings[i].bLgt:=1;
AllSettings[i].odValue.sValue[1]:=TmpItem.sValue[3];//0;
// Stop on Stall
i:=i+1;
CmpODRead(ENUM_SDO_2000.Aorta,	15,	ADR(TmpItem));
AllSettings[i].wIndex:=16#20A4;
AllSettings[i].bSubIndex:=2;
AllSettings[i].bLgt:=4;
AllSettings[i].odValue.dwValue:=TmpItem.dwValue;//85000;
// Homing Method
i:=i+1;
CmpODRead(ENUM_SDO_2000.Aorta,	12,	ADR(TmpItem));
AllSettings[i].wIndex:=16#6098;
AllSettings[i].bSubIndex:=0;
AllSettings[i].bLgt:=1;
AllSettings[i].odValue.sValue[1]:=TmpItem.sValue[4];//-2;
// Homing Acceleration
i:=i+1;
CmpODRead(ENUM_SDO_2000.Aorta,	16,	ADR(TmpItem));
AllSettings[i].wIndex:=16#609A;
AllSettings[i].bSubIndex:=0;
AllSettings[i].bLgt:=4;
AllSettings[i].odValue.dwValue:=TmpItem.dwValue;//341332;
// Homing Speeds Fast
i:=i+1;
CmpODRead(ENUM_SDO_2000.Aorta,	17,	ADR(TmpItem));
AllSettings[i].wIndex:=16#6099;
AllSettings[i].bSubIndex:=1;
AllSettings[i].bLgt:=4;
AllSettings[i].odValue.dwValue:=TmpItem.dwValue;//85333;
// Homing Speeds Slow
i:=i+1;
CmpODRead(ENUM_SDO_2000.Aorta,	18,	ADR(TmpItem));
AllSettings[i].wIndex:=16#6099;
AllSettings[i].bSubIndex:=2;
AllSettings[i].bLgt:=4;
AllSettings[i].odValue.dwValue:=TmpItem.dwValue;//85333;
//
// Positioning
//
// Position Window
i:=i+1;
CmpODRead(ENUM_SDO_2000.Aorta,	19,	ADR(TmpItem));
AllSettings[i].wIndex:=16#6067;
AllSettings[i].bSubIndex:=0;
AllSettings[i].bLgt:=4;
AllSettings[i].odValue.dwValue:=TmpItem.dwValue;//0;
// Profile Acceleration
i:=i+1;
CmpODRead(ENUM_SDO_2000.Aorta,	20,	ADR(TmpItem));
AllSettings[i].wIndex:=16#6083;
AllSettings[i].bSubIndex:=0;
AllSettings[i].bLgt:=4;
AllSettings[i].odValue.dwValue:=TmpItem.dwValue;//341332;
// Profile Deceleration
i:=i+1;
CmpODRead(ENUM_SDO_2000.Aorta,	21,	ADR(TmpItem));
AllSettings[i].wIndex:=16#6084;
AllSettings[i].bSubIndex:=0;
AllSettings[i].bLgt:=4;
AllSettings[i].odValue.dwValue:=TmpItem.dwValue;//341332;
// Profile Velocity
i:=i+1;
CmpODRead(ENUM_SDO_2000.Aorta,	22,	ADR(TmpItem));
AllSettings[i].wIndex:=16#6081;
AllSettings[i].bSubIndex:=0;
AllSettings[i].bLgt:=4;
AllSettings[i].odValue.dwValue:=TmpItem.dwValue;//85333;
// StallGuard Threshold
i:=i+1;
CmpODRead(ENUM_SDO_2000.Aorta,	23,	ADR(TmpItem));
AllSettings[i].wIndex:=16#209E;
AllSettings[i].bSubIndex:=1;
AllSettings[i].bLgt:=1;
AllSettings[i].odValue.sValue[1]:=TmpItem.sValue[1];//0;
// Stop on Stall
i:=i+1;
CmpODRead(ENUM_SDO_2000.Aorta,	24,	ADR(TmpItem));
AllSettings[i].wIndex:=16#20A4;
AllSettings[i].bSubIndex:=1;
AllSettings[i].bLgt:=4;
AllSettings[i].odValue.dwValue:=TmpItem.dwValue;//80000;
// only for version 2020-06-29
// Boost Current
i:=i+1;
CmpODRead(ENUM_SDO_2000.Aorta,	25,	ADR(TmpItem));
AllSettings[i].wIndex:=16#2006;
AllSettings[i].bSubIndex:=0;
AllSettings[i].bLgt:=1;
AllSettings[i].odValue.dwValue:=TmpItem.dwValue;//192;
// Boost Current Microsteps
i:=i+1;
CmpODRead(ENUM_SDO_2000.Aorta,	26,	ADR(TmpItem));
AllSettings[i].wIndex:=16#2007;
AllSettings[i].bSubIndex:=0;
AllSettings[i].bLgt:=4;
AllSettings[i].odValue.dwValue:=TmpItem.dwValue;//102400;

// set sync mode
i:=i+1;
AllSettings[i].wIndex:=16#1801;
AllSettings[i].bSubIndex:=2;
AllSettings[i].bLgt:=1;
AllSettings[i].odValue.dwValue:=11;//102400;


wNrSDO := i;
END_METHOD

METHOD mxGetSDO : BOOL;
VAR_INPUT
	wNr : WORD;
END_VAR
VAR_OUTPUT
	pTheSDO : pointer to SingleFullSDO;
END_VAR
IF wNr > wNrSDO THEN
	mxGetSDO:=FALSE;
	RETURN;	
END_IF
pTheSDO:=ADR(AllSettings[wNr]);
mxGetSDO:=TRUE;
END_METHOD

END_FUNCTION_BLOCK

// Aorta/AortaEngine/fbtAortaSettingsDownloader
FUNCTION_BLOCK fbtAortaSettingsDownloader IMPLEMENTS itf_settingsdownloader
VAR_INPUT
END_VAR
VAR_OUTPUT
END_VAR
VAR
	pLocDriver 			: POINTER TO fbtAorta_Trinamics; //_hardcodedsettings;
	fbAorta_Settings_1	: fbtAorta_AllSettings_Tri;
	fbAorta_Settings_2	: fbtAorta_AllSettings_Pri;
	xBusy 				: BOOL;
	strError 			: strDownloadError; // to avoid crashes

	xStartLoc 			: BOOL;
	eState				: ENUM_AortaDownloader_States;
	itfSelected 		: itf_SDO_FullList;
	dwVendorID			: DWORD;

END_VAR

METHOD mxDownload : BOOL
VAR_IN_OUT
	xStart : BOOL;
END_VAR
VAR_INPUT
	xAlways : BOOL;
END_VAR
VAR_OUTPUT
	xOK : BOOL;
END_VAR
IF xStart THEN
	xStart:=FALSE;
	xStartLoc := TRUE;
	eState := ENUM_AortaDownloader_States.findtype;
	xBusy:=TRUE;
	mxDownload := FALSE;
END_IF

CASE eState OF 
	ENUM_AortaDownloader_States.findtype :
		IF pLocDriver^.mxReadVendorID(xStart:=xStartLoc,dwVendorID=>dwVendorID, xOk=>xOk) THEN
			eState := ENUM_AortaDownloader_States.select;
		END_IF	
	
	ENUM_AortaDownloader_States.select :

		CASE dwVendorID OF
			16#286 : 	fbAorta_Settings_1.mxInit();
						itfSelected:=fbAorta_Settings_1; // trinamics

		ELSE 
			fbAorta_Settings_2.mxInit();
			itfSelected:=fbAorta_Settings_2;
		END_CASE
		xStartLoc := TRUE;
		eState := ENUM_AortaDownloader_States.download;
	
	ENUM_AortaDownloader_States.download :

		IF	pLocDriver^.mxDumpSettings(xStart := xStartLoc, itfSettings := itfSelected,	xOk => xOk)	THEN
			mxDownload := TRUE;
			xBusy:=FALSE;
		END_IF

END_CASE
END_METHOD

PROPERTY PUBLIC prpbActiveSubIndex : BYTE
GET
END_GET
END_PROPERTY

PROPERTY prpbStatus : eDownloaderResults
SET
END_SET
GET
END_GET
END_PROPERTY

PROPERTY PUBLIC prpxBusy : BOOL
GET
prpxBusy := xBusy;
END_GET
END_PROPERTY

METHOD mxInit : BOOL
VAR_INPUT
	pDriver : POINTER TO fbtAorta_Trinamics; //_hardcodedsettings;
END_VAR
pLocDriver:=pDriver;
END_METHOD

PROPERTY prppDownloadError : pointer to strDownloadError
GET
prppDownloadError:=ADR(strError);
END_GET
END_PROPERTY

END_FUNCTION_BLOCK

// Aorta/Driver/Settings/fbtAorta_AllSettings_Pri
FUNCTION_BLOCK fbtAorta_AllSettings_Pri EXTENDS fbtSDO_FullList_Base 
VAR_INPUT
END_VAR
VAR_OUTPUT
END_VAR
VAR
	AllSettings : ARRAY[1..25] OF SingleFullSDO;
END_VAR

METHOD mxAdd : BOOL
VAR_INPUT
	wOD_Idx   : WORD; // location in OD
	wOD_SIx   : BYTE; // location in OD
	wIndex    : WORD;
	wSubIndex : BYTE;
	bLength   : BYTE;
	bPosition : BYTE;
END_VAR
VAR_IN_OUT
	i : WORD;
END_VAR
VAR
	TmpItem	: ODItem;
END_VAR
CmpODRead(wOD_Idx,	wOD_SIx,	ADR(TmpItem));
AllSettings[i].wIndex:=wIndex;
AllSettings[i].bSubIndex:=wSubIndex;
AllSettings[i].bLgt:=bLength;
CASE bLength OF
	1 : AllSettings[i].odValue.sValue[1]:=TmpItem.sValue[bPosition];
	2 : AllSettings[i].odValue.wValue[1]:=TmpItem.wValue[bPosition];
	4 : AllSettings[i].odValue.dwValue:=TmpItem.dwValue;
END_CASE
i:=i+1;
END_METHOD

METHOD mxGetSDO : BOOL;
VAR_INPUT
	wNr : WORD;
END_VAR
VAR_OUTPUT
	pTheSDO : pointer to SingleFullSDO;
END_VAR
IF wNr > wNrSDO THEN
	mxGetSDO:=FALSE;
	RETURN;	
END_IF
pTheSDO:=ADR(AllSettings[wNr]);
mxGetSDO:=TRUE;
END_METHOD

METHOD mxInit : BOOL
VAR_INPUT
END_VAR
VAR
	i : WORD;
	TmpItem	: ODItem;
END_VAR
i:=1;
SysMemSet(ADR(AllSettings),0,SIZEOF(AllSettings));
mxAdd(wOD_Idx:=ENUM_SDO_2000.Aorta,wOD_SIx:=27,bLength:=1,bPosition:=4,wIndex:=16#6098,wSubIndex:=0,i:=i);
mxAdd(wOD_Idx:=ENUM_SDO_2000.Aorta,wOD_SIx:=28,bLength:=4,bPosition:=0,wIndex:=16#609A,wSubIndex:=0,i:=i);
mxAdd(wOD_Idx:=ENUM_SDO_2000.Aorta,wOD_SIx:=29,bLength:=4,bPosition:=0,wIndex:=16#6099,wSubIndex:=1,i:=i);
mxAdd(wOD_Idx:=ENUM_SDO_2000.Aorta,wOD_SIx:=30,bLength:=4,bPosition:=0,wIndex:=16#6099,wSubIndex:=2,i:=i);
mxAdd(wOD_Idx:=ENUM_SDO_2000.Aorta,wOD_SIx:=31,bLength:=4,bPosition:=0,wIndex:=16#6067,wSubIndex:=0,i:=i);
mxAdd(wOD_Idx:=ENUM_SDO_2000.Aorta,wOD_SIx:=32,bLength:=4,bPosition:=0,wIndex:=16#6083,wSubIndex:=0,i:=i);
mxAdd(wOD_Idx:=ENUM_SDO_2000.Aorta,wOD_SIx:=33,bLength:=4,bPosition:=0,wIndex:=16#6084,wSubIndex:=0,i:=i);
mxAdd(wOD_Idx:=ENUM_SDO_2000.Aorta,wOD_SIx:=34,bLength:=4,bPosition:=0,wIndex:=16#6081,wSubIndex:=0,i:=i);
wNrSDO := i;
END_METHOD

END_FUNCTION_BLOCK

// Aorta/Special Alarm/fbtProtecSpec_STCValve
FUNCTION_BLOCK fbtProtecSpec_STCValve EXTENDS fbtBaseSpecialProtection
VAR
	fbProtectionInfo				: fbtProtecSpec_STCValve_Info;
	itfSTCValve						: itf_STCValve;
	xActive							: BOOL;
	tDelay							: TIME;
	xAlarmCondition					: BOOL;
	bType							: BYTE;
	ShutdownLatch 					: SR;
	ResettableWarning				: SR;
	bStallsCounter					: BYTE	:= 0;
	fbDelayAtStart_AtSignal			: fbtDelayAtStart_AtSignal;
	bDelay							: BYTE;
END_VAR
VAR CONSTANT
	bStallsBeforeTrigger			: BYTE	:= 3;
END_VAR

METHOD mxInitSpecial : BOOL
VAR_INPUT
	wNameIn					: WORD;
	wSDOIn					: WORD;
	itfSTCValveIn			: itf_STCValve;
END_VAR
VAR
	itfProtecPermisSystem	: itf_ProtecPermisSystem;
	itfListProtections		: itf_ListProtections;
	itfLocalRoot			: itf_SystemRoot;
END_VAR
mxInitSpecial := TRUE;
xActive := TRUE;

IF NOT __QUERYINTERFACE(GVL_itfRoot,	itfLocalRoot) THEN	RETURN;	END_IF

itfSTCValve := itfSTCValveIn;

itfProtecPermisSystem	:= itfLocalRoot.prpitfProtecPermisSystem;
IF 	itfProtecPermisSystem	= 0 THEN	mxInitSpecial := FALSE;	RETURN;	END_IF
itfListProtections	:= itfProtecPermisSystem.prpitfProtectionsSpecial;
IF itfListProtections = 0 THEN	mxInitSpecial := FALSE;	RETURN;	END_IF

wName					:= wNameIn;
wSDOIndex				:= wSDOIn;

fbProtectionInfo.mInit(itfSTCValveIn);

mxInit(wSDOIndex);

IF THIS^.mxExists() THEN
	mxInitSpecial:=itfListProtections.mxAddProtection(THIS^);
ELSE
	mxInitSpecial := THIS^.mxLoadSettings();
	mxInitSpecial := itfListProtections.mxAddProtection_Base(THIS^);	
END_IF
END_METHOD

METHOD mxLoadSettings : BOOL
VAR
	tmpOD	: ODItem;
	b		: BYTE;
END_VAR
mxLoadSettings	:= TRUE;
IF NOT CmpODRead(wSDOIndex,	1,	ADR(tmpOD)) OR itfSTCValve = 0 THEN RETURN; END_IF
xActive	:= tmpOD.xValue[1];
IF NOT xActive THEN  RETURN; END_IF
CmpODRead(wSDOIndex,	2,	ADR(tmpOD));
bType := tmpOD.bValue[1];
bDelay := LIMIT(tmpOD.bValue[4], tmpOD.bValue[3], tmpOD.bValue[2]);
END_METHOD

METHOD mwCheckProtection : WORD
VAR_INPUT
	itfStatusInfo	: itf_StatusInfo;
END_VAR
VAR
	wError					: WORD;
	_xAlarmCond_PreWarning	: BOOL;
	_xAlarmCond_Warning		: BOOL;
	_xAlarmCond_Shutdown	: BOOL;
	_xAlarmCond_ResetWarn	: BOOL;
	xAlarmConditionTemp		: BOOL;
	xTimerTriggered			: BOOL;
	//xResult			: BOOL;
	//xTrigger		: BOOL;
	//wIndex  		: WORD;
END_VAR
IF NOT xActive THEN
	wError := Aorta_Errors.STCValve_Active_No_Alarm;
	itfSTCValve.prpwError := Aorta_Errors.STCValve_Active_No_Alarm;
ELSE
	wError := itfSTCValve.prpwError;	
END_IF

xAlarmConditionTemp := wError<>0;

IF xActive THEN
	IF wError = Aorta_Errors.CAN_Out THEN
		_xAlarmCond_Shutdown	:= TRUE;		
	ELSE
		IF wError = Aorta_Errors.Position_Stall AND bStallsCounter < bStallsBeforeTrigger THEN
			bStallsCounter := bStallsCounter + 1;
		END_IF
		IF wError<>Aorta_Errors.Position_Stall OR bStallsCounter >= bStallsBeforeTrigger THEN
			_xAlarmCond_PreWarning	:= bType.0 AND xAlarmConditionTemp;
			_xAlarmCond_Warning		:= bType.1 AND xAlarmConditionTemp;
			_xAlarmCond_Shutdown	:= bType.2 AND xAlarmConditionTemp;
			_xAlarmCond_ResetWarn	:= bType.3 AND xAlarmConditionTemp;
		ELSE
			itfSTCValve.prpwError := 0;	
		END_IF
	END_IF
ELSE
	_xAlarmCond_Warning		:= TRUE;
END_IF

xAlarmCondition := _xAlarmCond_PreWarning OR _xAlarmCond_Warning OR _xAlarmCond_Shutdown OR _xAlarmCond_ResetWarn;
xTimerTriggered := fbDelayAtStart_AtSignal.mxRun(0, 0, bDelay, xAlarmCondition);

ResettableWarning(Set1:=xTimerTriggered AND _xAlarmCond_ResetWarn, Reset := FALSE);
ShutdownLatch(Set1:=xTimerTriggered AND _xAlarmCond_Shutdown, Reset:=FALSE);

//protection triggered => set the correct bit
theStatus.wValue[1].0 := _xAlarmCond_PreWarning	AND xTimerTriggered;
theStatus.wValue[1].1 := (_xAlarmCond_Warning	AND xTimerTriggered) OR ResettableWarning.Q1;
theStatus.wValue[1].3 := ShutdownLatch.Q1;

mwCheckProtection:=SUPER^.mwCheckProtection(itfStatusInfo);

//Fill 3000 Data
dw3000Data:=wSDOIndex;
dw3000Data:=SHL(dw3000Data,16) OR theStatus.wValue[1];
END_METHOD

PROPERTY prpitfProtectionInfo : itf_protectioninfo
GET
prpitfProtectionInfo := fbProtectionInfo;
END_GET
END_PROPERTY

PROPERTY prpxMoreInfo : BOOL
GET
{IF defined (Mk5S_Touch)}
prpxMoreInfo	:= TRUE;
{ELSE}
prpxMoreInfo	:= FALSE;
{END_IF}
END_GET
END_PROPERTY

METHOD mxReset : BOOL
VAR_INPUT
	itfStatusInfo 	: itf_statusinfo;
	xProtection 	: BOOL;
	xService		: BOOL;
END_VAR
VAR
	wError 			: WORD;
END_VAR
mxReset := FALSE;

IF  xAlarmCondition THEN
	itfSTCValve.mReset();
	bStallsCounter := 0;
	ResettableWarning(Set1:=FALSE, RESET := TRUE);
	ShutdownLatch(Set1:=FALSE, RESET:=TRUE);
	fbDelayAtStart_AtSignal.mReset();
	mxReset	:= TRUE;
END_IF
END_METHOD

METHOD mxResolveMPLLinks : BOOL
VAR_INPUT
	MPLList : itf_MPLList;
	IVLList : itf_IVLList;
END_VAR
mxResolveMPLLinks:=TRUE;
END_METHOD

END_FUNCTION_BLOCK

// Aorta/Special Alarm/fbtProtecSpec_STCValve_Info
FUNCTION_BLOCK fbtProtecSpec_STCValve_Info IMPLEMENTS itf_ProtectionInfo
VAR
	itfSTCValve		: itf_STCValve;
END_VAR

